LIN {X 0,Y 569.296,Z 343.315,A -85,B 0,C 180,E1 25931.653,E2 25931.653} C_VEL
LIN {X 0,Y 569.324,Z 343.315,A -85,B 0,C 180,E1 25928.382,E2 25928.382} C_VEL
LIN {X 0,Y 569.296,Z 343.305,A -85,B 0,C 180,E1 25925.543,E2 25925.543} C_VEL
LIN {X 0,Y 569.333,Z 343.299,A -85,B 0,C 180,E1 25922.315,E2 25922.315} C_VEL
LIN {X 0,Y 569.297,Z 343.304,A -85,B 0,C 180,E1 25919.396,E2 25919.396} C_VEL
LIN {X 0,Y 569.337,Z 343.298,A -85,B 0,C 180,E1 25916.173,E2 25916.173} C_VEL
LIN {X 0,Y 569.304,Z 343.315,A -85,B 0,C 180,E1 25913.141,E2 25913.141} C_VEL
LIN {X 0,Y 569.317,Z 343.31,A -85,B 0,C 180,E1 25909.782,E2 25909.782} C_VEL
LIN {X 0,Y 569.309,Z 343.253,A -85,B 0,C 180,E1 25906.802,E2 25906.802} C_VEL
LIN {X 0,Y 569.309,Z 343.313,A -85,B 0,C 180,E1 25903.47,E2 25903.47} C_VEL
LIN {X 0,Y 569.334,Z 343.255,A -85,B 0,C 180,E1 25900.4,E2 25900.4} C_VEL
LIN {X 0,Y 569.305,Z 343.303,A -85,B 0,C 180,E1 25897.226,E2 25897.226} C_VEL
LIN {X 0,Y 569.343,Z 343.264,A -85,B 0,C 180,E1 25894.18,E2 25894.18} C_VEL
LIN {X 0,Y 569.305,Z 343.306,A -85,B 0,C 180,E1 25891,E2 25891} C_VEL
LIN {X 0,Y 569.313,Z 343.38,A -85,B 0,C 180,E1 25890.889,E2 25890.889} C_VEL
LIN {X 0,Y 570.615,Z 346.769,A -85,B 0,C 180,E1 25890.271,E2 25890.271} C_VEL
LIN {X 0,Y 571.971,Z 348.701,A -85,B 0,C 180,E1 25889.828,E2 25889.828} C_VEL
LIN {X 0,Y 574.926,Z 352.956,A -85,B 0,C 180,E1 25889.248,E2 25889.248} C_VEL
LIN {X 0,Y 584.169,Z 364.72,A -85,B 0,C 180,E1 25887.634,E2 25887.634} C_VEL
LIN {X 0,Y 598.802,Z 384.338,A -85,B 0,C 180,E1 25885.262,E2 25885.262} C_VEL
LIN {X 0,Y 616.624,Z 409.316,A -85,B 0,C 180,E1 25882.622,E2 25882.622} C_VEL
LIN {X 0,Y 624.459,Z 421.118,A -85,B 0,C 180,E1 25881.519,E2 25881.519} C_VEL
LIN {X 0,Y 618.445,Z 624.42,A -85,B 0,C 180,E1 25878.613,E2 25878.613} C_VEL
LIN {X 0,Y 612.62,Z 826.414,A -85,B 0,C 180,E1 25875.768,E2 25875.768} C_VEL
LIN {X 0,Y 611.271,Z 850.143,A -85,B 0,C 180,E1 25875.338,E2 25875.338} C_VEL
LIN {X 0,Y 609.033,Z 878.867,A -85,B 0,C 180,E1 25874.632,E2 25874.632} C_VEL
LIN {X 0,Y 606.973,Z 900.534,A -85,B 0,C 180,E1 25873.955,E2 25873.955} C_VEL
LIN {X 0,Y 604.712,Z 921.393,A -85,B 0,C 180,E1 25873.181,E2 25873.181} C_VEL
LIN {X 0,Y 602.472,Z 940.413,A -85,B 0,C 180,E1 25872.36,E2 25872.36} C_VEL
LIN {X 0,Y 599.944,Z 959.81,A -85,B 0,C 180,E1 25871.41,E2 25871.41} C_VEL
LIN {X 0,Y 597.096,Z 980.312,A -85,B 0,C 180,E1 25870.268,E2 25870.268} C_VEL
LIN {X 0,Y 593.449,Z 1004.907,A -85,B 0,C 180,E1 25868.687,E2 25868.687} C_VEL
LIN {X 0,Y 590.181,Z 1025.558,A -85,B 0,C 180,E1 25867.154,E2 25867.154} C_VEL
LIN {X 0,Y 587.381,Z 1042.97,A -85,B 0,C 180,E1 25865.709,E2 25865.709} C_VEL
LIN {X 0,Y 584.6,Z 1060.165,A -85,B 0,C 180,E1 25864.124,E2 25864.124} C_VEL
LIN {X 0,Y 581.463,Z 1079.875,A -85,B 0,C 180,E1 25862.096,E2 25862.096} C_VEL
LIN {X 0,Y 578.616,Z 1097.987,A -85,B 0,C 180,E1 25859.96,E2 25859.96} C_VEL
LIN {X 0,Y 576.364,Z 1112.967,A -85,B 0,C 180,E1 25857.99,E2 25857.99} C_VEL
LIN {X 0,Y 574.256,Z 1127.882,A -85,B 0,C 180,E1 25855.803,E2 25855.803} C_VEL
LIN {X 0,Y 572.235,Z 1143.703,A -85,B 0,C 180,E1 25853.15,E2 25853.15} C_VEL
LIN {X 0,Y 570.92,Z 1155.266,A -85,B 0,C 180,E1 25850.932,E2 25850.932} C_VEL
LIN {X 0,Y 569.924,Z 1165.445,A -85,B 0,C 180,E1 25848.726,E2 25848.726} C_VEL
LIN {X 0,Y 569.029,Z 1176.304,A -85,B 0,C 180,E1 25846.015,E2 25846.015} C_VEL
LIN {X 0,Y 568.479,Z 1185.17,A -85,B 0,C 180,E1 25843.321,E2 25843.321} C_VEL
LIN {X 0,Y 568.159,Z 1191.597,A -85,B 0,C 180,E1 25840.956,E2 25840.956} C_VEL
LIN {X 0,Y 568.007,Z 1197.191,A -85,B 0,C 180,E1 25838.381,E2 25838.381} C_VEL
LIN {X 0,Y 567.933,Z 1201.538,A -85,B 0,C 180,E1 25835.557,E2 25835.557} C_VEL
LIN {X 0,Y 567.917,Z 1203.848,A -85,B 0,C 180,E1 25833.129,E2 25833.129} C_VEL
LIN {X 0,Y 567.906,Z 1204.804,A -85,B 0,C 180,E1 25830.908,E2 25830.908} C_VEL
LIN {X 0,Y 567.916,Z 1204.736,A -85,B 0,C 180,E1 25828.789,E2 25828.789} C_VEL
LIN {X 0,Y 567.912,Z 1203.507,A -85,B 0,C 180,E1 25826.366,E2 25826.366} C_VEL
LIN {X 0,Y 567.948,Z 1200.336,A -85,B 0,C 180,E1 25823.531,E2 25823.531} C_VEL
LIN {X 0,Y 568.029,Z 1196.126,A -85,B 0,C 180,E1 25821.089,E2 25821.089} C_VEL
LIN {X 0,Y 568.191,Z 1190.834,A -85,B 0,C 180,E1 25818.736,E2 25818.736} C_VEL
LIN {X 0,Y 568.577,Z 1183.471,A -85,B 0,C 180,E1 25816.106,E2 25816.106} C_VEL
LIN {X 0,Y 569.205,Z 1173.921,A -85,B 0,C 180,E1 25813.362,E2 25813.362} C_VEL
LIN {X 0,Y 570.006,Z 1164.53,A -85,B 0,C 180,E1 25811.064,E2 25811.064} C_VEL
LIN {X 0,Y 571.043,Z 1154.241,A -85,B 0,C 180,E1 25808.857,E2 25808.857} C_VEL
LIN {X 0,Y 572.616,Z 1140.8,A -85,B 0,C 180,E1 25806.321,E2 25806.321} C_VEL
LIN {X 0,Y 574.531,Z 1125.781,A -85,B 0,C 180,E1 25803.877,E2 25803.877} C_VEL
LIN {X 0,Y 576.537,Z 1111.839,A -85,B 0,C 180,E1 25801.854,E2 25801.854} C_VEL
LIN {X 0,Y 579.026,Z 1095.326,A -85,B 0,C 180,E1 25799.704,E2 25799.704} C_VEL
LIN {X 0,Y 582.167,Z 1075.37,A -85,B 0,C 180,E1 25797.428,E2 25797.428} C_VEL
LIN {X 0,Y 584.781,Z 1059.05,A -85,B 0,C 180,E1 25795.77,E2 25795.77} C_VEL
LIN {X 0,Y 587.479,Z 1042.377,A -85,B 0,C 180,E1 25794.24,E2 25794.24} C_VEL
LIN {X 0,Y 590.375,Z 1024.364,A -85,B 0,C 180,E1 25792.752,E2 25792.752} C_VEL
LIN {X 0,Y 594.048,Z 1001.028,A -85,B 0,C 180,E1 25791.044,E2 25791.044} C_VEL
LIN {X 0,Y 597.217,Z 979.404,A -85,B 0,C 180,E1 25789.679,E2 25789.679} C_VEL
LIN {X 0,Y 599.973,Z 959.579,A -85,B 0,C 180,E1 25788.578,E2 25788.578} C_VEL
LIN {X 0,Y 602.469,Z 940.393,A -85,B 0,C 180,E1 25787.639,E2 25787.639} C_VEL
LIN {X 0,Y 604.747,Z 921.017,A -85,B 0,C 180,E1 25786.805,E2 25786.805} C_VEL
LIN {X 0,Y 607.067,Z 899.553,A -85,B 0,C 180,E1 25786.013,E2 25786.013} C_VEL
LIN {X 0,Y 609.581,Z 872.863,A -85,B 0,C 180,E1 25785.2,E2 25785.2} C_VEL
LIN {X 0,Y 611.435,Z 847.126,A -85,B 0,C 180,E1 25784.602,E2 25784.602} C_VEL
LIN {X 0,Y 612.671,Z 825.024,A -85,B 0,C 180,E1 25784.212,E2 25784.212} C_VEL
LIN {X 0,Y 618.765,Z 612.923,A -85,B 0,C 180,E1 25781.224,E2 25781.224} C_VEL
LIN {X 0,Y 624.762,Z 420.905,A -85,B 0,C 180,E1 25778.456,E2 25778.456} C_VEL
LIN {X 0,Y 613.339,Z 403.227,A -85,B 0,C 180,E1 25776.668,E2 25776.668} C_VEL
LIN {X 0,Y 604.018,Z 389.622,A -85,B 0,C 180,E1 25775.088,E2 25775.088} C_VEL
LIN {X 0,Y 597.282,Z 380.633,A -85,B 0,C 180,E1 25773.881,E2 25773.881} C_VEL
LIN {X 0,Y 592.482,Z 374.303,A -85,B 0,C 180,E1 25772.974,E2 25772.974} C_VEL
LIN {X 0,Y 588.914,Z 369.679,A -85,B 0,C 180,E1 25772.274,E2 25772.274} C_VEL
LIN {X 0,Y 581.287,Z 359.993,A -85,B 0,C 180,E1 25770.694,E2 25770.694} C_VEL
LIN {X 0,Y 577.779,Z 355.627,A -85,B 0,C 180,E1 25769.923,E2 25769.923} C_VEL
LIN {X 0,Y 576.035,Z 353.726,A -85,B 0,C 180,E1 25769.536,E2 25769.536} C_VEL
LIN {X 0,Y 572.86,Z 349.891,A -85,B 0,C 180,E1 25768.799,E2 25768.799} C_VEL
LIN {X 0,Y 571.886,Z 348.208,A -85,B 0,C 180,E1 25768.51,E2 25768.51} C_VEL
LIN {X 0,Y 569.602,Z 344.596,A -85,B 0,C 180,E1 25767.495,E2 25767.495} C_VEL
LIN {X 0,Y 569.31,Z 343.269,A -85,B 0,C 180,E1 25767.171,E2 25767.171} C_VEL
LIN {X 0,Y 569.38,Z 343.289,A -85,B 0,C 180,E1 25764.043,E2 25764.043} C_VEL
LIN {X 0,Y 569.313,Z 343.291,A -85,B 0,C 180,E1 25760.881,E2 25760.881} C_VEL
LIN {X 0,Y 569.371,Z 343.26,A -85,B 0,C 180,E1 25757.687,E2 25757.687} C_VEL
LIN {X 0,Y 569.319,Z 343.314,A -85,B 0,C 180,E1 25754.546,E2 25754.546} C_VEL
LIN {X 0,Y 569.347,Z 343.269,A -85,B 0,C 180,E1 25751.241,E2 25751.241} C_VEL
LIN {X 0,Y 569.32,Z 343.289,A -85,B 0,C 180,E1 25748.28,E2 25748.28} C_VEL
LIN {X 0,Y 569.338,Z 343.294,A -85,B 0,C 180,E1 25744.937,E2 25744.937} C_VEL
LIN {X 0,Y 569.33,Z 343.268,A -85,B 0,C 180,E1 25741.912,E2 25741.912} C_VEL
LIN {X 0,Y 569.33,Z 343.315,A -85,B 0,C 180,E1 25738.591,E2 25738.591} C_VEL
LIN {X 0,Y 569.357,Z 343.259,A -85,B 0,C 180,E1 25735.467,E2 25735.467} C_VEL
LIN {X 0,Y 569.322,Z 343.3,A -85,B 0,C 180,E1 25732.228,E2 25732.228} C_VEL
LIN {X 0,Y 569.379,Z 343.279,A -85,B 0,C 180,E1 25729,E2 25729} C_VEL
LIN {X 0,Y 569.319,Z 343.267,A -85,B 0,C 180,E1 25725.799,E2 25725.799} C_VEL
LIN {X 0,Y 569.368,Z 343.301,A -85,B 0,C 180,E1 25722.524,E2 25722.524} C_VEL
LIN {X 0,Y 569.329,Z 343.284,A -85,B 0,C 180,E1 25719.399,E2 25719.399} C_VEL
LIN {X 0,Y 569.392,Z 343.421,A -85,B 0,C 180,E1 25718.9,E2 25718.9} C_VEL
LIN {X 0,Y 570.358,Z 346.246,A -85,B 0,C 180,E1 25718.614,E2 25718.614} C_VEL
LIN {X 0,Y 572.684,Z 348.869,A -85,B 0,C 180,E1 25718.06,E2 25718.06} C_VEL
LIN {X 0,Y 574.711,Z 350.146,A -85,B 0,C 180,E1 25717.617,E2 25717.617} C_VEL
LIN {X 0,Y 576.858,Z 353.718,A -85,B 0,C 180,E1 25717.099,E2 25717.099} C_VEL
LIN {X 0,Y 580.018,Z 356.535,A -85,B 0,C 180,E1 25716.425,E2 25716.425} C_VEL
LIN {X 0,Y 582.778,Z 360.473,A -85,B 0,C 180,E1 25715.818,E2 25715.818} C_VEL
LIN {X 0,Y 585.289,Z 362.868,A -85,B 0,C 180,E1 25715.311,E2 25715.311} C_VEL
LIN {X 0,Y 588.636,Z 367.172,A -85,B 0,C 180,E1 25714.628,E2 25714.628} C_VEL
LIN {X 0,Y 597.326,Z 377.95,A -85,B 0,C 180,E1 25712.969,E2 25712.969} C_VEL
LIN {X 0,Y 608.831,Z 393.554,A -85,B 0,C 180,E1 25710.941,E2 25710.941} C_VEL
LIN {X 0,Y 620.103,Z 410.5,A -85,B 0,C 180,E1 25709.111,E2 25709.111} C_VEL
LIN {X 0,Y 624.682,Z 417.785,A -85,B 0,C 180,E1 25708.41,E2 25708.41} C_VEL
LIN {X 0,Y 618.203,Z 625.916,A -85,B 0,C 180,E1 25705.412,E2 25705.412} C_VEL
LIN {X 0,Y 614.777,Z 746.22,A -85,B 0,C 180,E1 25703.721,E2 25703.721} C_VEL
LIN {X 0,Y 613.881,Z 753.921,A -85,B 0,C 180,E1 25703.681,E2 25703.681} C_VEL
LIN {X 0,Y 608.994,Z 774.548,A -85,B 0,C 180,E1 25703.822,E2 25703.822} C_VEL
LIN {X 0,Y 608.288,Z 781.156,A -85,B 0,C 180,E1 25703.781,E2 25703.781} C_VEL
LIN {X 0,Y 606.727,Z 825.165,A -85,B 0,C 180,E1 25703.134,E2 25703.134} C_VEL
LIN {X 0,Y 604.843,Z 852.015,A -85,B 0,C 180,E1 25702.575,E2 25702.575} C_VEL
LIN {X 0,Y 602.85,Z 874.745,A -85,B 0,C 180,E1 25701.965,E2 25701.965} C_VEL
LIN {X 0,Y 600.188,Z 900.951,A -85,B 0,C 180,E1 25701.092,E2 25701.092} C_VEL
LIN {X 0,Y 597.063,Z 926.428,A -85,B 0,C 180,E1 25700.042,E2 25700.042} C_VEL
LIN {X 0,Y 593.864,Z 950.106,A -85,B 0,C 180,E1 25698.888,E2 25698.888} C_VEL
LIN {X 0,Y 590.327,Z 973.89,A -85,B 0,C 180,E1 25697.529,E2 25697.529} C_VEL
LIN {X 0,Y 587.148,Z 993.791,A -85,B 0,C 180,E1 25696.222,E2 25696.222} C_VEL
LIN {X 0,Y 583.963,Z 1013.149,A -85,B 0,C 180,E1 25694.794,E2 25694.794} C_VEL
LIN {X 0,Y 580.163,Z 1035.792,A -85,B 0,C 180,E1 25692.902,E2 25692.902} C_VEL
LIN {X 0,Y 576.836,Z 1055.052,A -85,B 0,C 180,E1 25691.059,E2 25691.059} C_VEL
LIN {X 0,Y 573.849,Z 1072.78,A -85,B 0,C 180,E1 25689.16,E2 25689.16} C_VEL
LIN {X 0,Y 570.546,Z 1092.991,A -85,B 0,C 180,E1 25686.697,E2 25686.697} C_VEL
LIN {X 0,Y 568.077,Z 1108.692,A -85,B 0,C 180,E1 25684.523,E2 25684.523} C_VEL
LIN {X 0,Y 565.787,Z 1124.739,A -85,B 0,C 180,E1 25682.016,E2 25682.016} C_VEL
LIN {X 0,Y 563.914,Z 1138.861,A -85,B 0,C 180,E1 25679.47,E2 25679.47} C_VEL
LIN {X 0,Y 562.473,Z 1151.648,A -85,B 0,C 180,E1 25676.841,E2 25676.841} C_VEL
LIN {X 0,Y 561.38,Z 1163.044,A -85,B 0,C 180,E1 25674.071,E2 25674.071} C_VEL
LIN {X 0,Y 560.732,Z 1171.84,A -85,B 0,C 180,E1 25671.551,E2 25671.551} C_VEL
LIN {X 0,Y 560.291,Z 1179.722,A -85,B 0,C 180,E1 25668.844,E2 25668.844} C_VEL
LIN {X 0,Y 560.05,Z 1185.816,A -85,B 0,C 180,E1 25666.152,E2 25666.152} C_VEL
LIN {X 0,Y 559.953,Z 1189.82,A -85,B 0,C 180,E1 25663.844,E2 25663.844} C_VEL
LIN {X 0,Y 559.917,Z 1192.912,A -85,B 0,C 180,E1 25661.328,E2 25661.328} C_VEL
LIN {X 0,Y 559.909,Z 1194.644,A -85,B 0,C 180,E1 25658.627,E2 25658.627} C_VEL
LIN {X 0,Y 559.913,Z 1194.855,A -85,B 0,C 180,E1 25656.254,E2 25656.254} C_VEL
LIN {X 0,Y 559.91,Z 1193.988,A -85,B 0,C 180,E1 25653.994,E2 25653.994} C_VEL
LIN {X 0,Y 559.923,Z 1191.789,A -85,B 0,C 180,E1 25651.535,E2 25651.535} C_VEL
LIN {X 0,Y 560.002,Z 1187.772,A -85,B 0,C 180,E1 25648.772,E2 25648.772} C_VEL
LIN {X 0,Y 560.145,Z 1182.479,A -85,B 0,C 180,E1 25646.213,E2 25646.213} C_VEL
LIN {X 0,Y 560.447,Z 1176.363,A -85,B 0,C 180,E1 25643.855,E2 25643.855} C_VEL
LIN {X 0,Y 560.961,Z 1168.311,A -85,B 0,C 180,E1 25641.286,E2 25641.286} C_VEL
LIN {X 0,Y 561.873,Z 1157.755,A -85,B 0,C 180,E1 25638.504,E2 25638.504} C_VEL
LIN {X 0,Y 562.987,Z 1146.754,A -85,B 0,C 180,E1 25636.023,E2 25636.023} C_VEL
LIN {X 0,Y 564.674,Z 1132.973,A -85,B 0,C 180,E1 25633.331,E2 25633.331} C_VEL
LIN {X 0,Y 566.562,Z 1118.874,A -85,B 0,C 180,E1 25630.945,E2 25630.945} C_VEL
LIN {X 0,Y 568.991,Z 1103.007,A -85,B 0,C 180,E1 25628.561,E2 25628.561} C_VEL
LIN {X 0,Y 571.836,Z 1084.833,A -85,B 0,C 180,E1 25626.178,E2 25626.178} C_VEL
LIN {X 0,Y 574.666,Z 1067.976,A -85,B 0,C 180,E1 25624.217,E2 25624.217} C_VEL
LIN {X 0,Y 578.197,Z 1047.445,A -85,B 0,C 180,E1 25622.091,E2 25622.091} C_VEL
LIN {X 0,Y 581.602,Z 1027.065,A -85,B 0,C 180,E1 25620.25,E2 25620.25} C_VEL
LIN {X 0,Y 584.696,Z 1008.633,A -85,B 0,C 180,E1 25618.766,E2 25618.766} C_VEL
LIN {X 0,Y 588.482,Z 985.63,A -85,B 0,C 180,E1 25617.123,E2 25617.123} C_VEL
LIN {X 0,Y 591.988,Z 962.709,A -85,B 0,C 180,E1 25615.718,E2 25615.718} C_VEL
LIN {X 0,Y 595.353,Z 939.327,A -85,B 0,C 180,E1 25614.473,E2 25614.473} C_VEL
LIN {X 0,Y 598.747,Z 912.783,A -85,B 0,C 180,E1 25613.282,E2 25613.282} C_VEL
LIN {X 0,Y 601.432,Z 889.096,A -85,B 0,C 180,E1 25612.402,E2 25612.402} C_VEL
LIN {X 0,Y 604.11,Z 861.148,A -85,B 0,C 180,E1 25611.56,E2 25611.56} C_VEL
LIN {X 0,Y 605.996,Z 835.793,A -85,B 0,C 180,E1 25610.979,E2 25610.979} C_VEL
LIN {X 0,Y 607.3,Z 812.342,A -85,B 0,C 180,E1 25610.575,E2 25610.575} C_VEL
LIN {X 0,Y 613.778,Z 596.837,A -85,B 0,C 180,E1 25607.52,E2 25607.52} C_VEL
LIN {X 0,Y 619.14,Z 421.569,A -85,B 0,C 180,E1 25604.997,E2 25604.997} C_VEL
LIN {X 0,Y 605.811,Z 402.395,A -85,B 0,C 180,E1 25603.07,E2 25603.07} C_VEL
LIN {X 0,Y 589.286,Z 379.992,A -85,B 0,C 180,E1 25600.5,E2 25600.5} C_VEL
LIN {X 0,Y 583.743,Z 372.893,A -85,B 0,C 180,E1 25599.583,E2 25599.583} C_VEL
LIN {X 0,Y 579.056,Z 367.062,A -85,B 0,C 180,E1 25598.784,E2 25598.784} C_VEL
LIN {X 0,Y 575.08,Z 362.1,A -85,B 0,C 180,E1 25598.083,E2 25598.083} C_VEL
LIN {X 0,Y 571.76,Z 358.178,A -85,B 0,C 180,E1 25597.487,E2 25597.487} C_VEL
LIN {X 0,Y 570.576,Z 356.419,A -85,B 0,C 180,E1 25597.262,E2 25597.262} C_VEL
LIN {X 0,Y 567.534,Z 353.373,A -85,B 0,C 180,E1 25596.709,E2 25596.709} C_VEL
LIN {X 0,Y 565.807,Z 350.517,A -85,B 0,C 180,E1 25596.363,E2 25596.363} C_VEL
LIN {X 0,Y 563.016,Z 348.232,A -85,B 0,C 180,E1 25595.847,E2 25595.847} C_VEL
LIN {X 0,Y 561.6,Z 345.253,A -85,B 0,C 180,E1 25595.537,E2 25595.537} C_VEL
LIN {X 0,Y 561.418,Z 344.297,A -85,B 0,C 180,E1 25595.455,E2 25595.455} C_VEL
LIN {X 0,Y 561.348,Z 344.296,A -85,B 0,C 180,E1 25592.301,E2 25592.301} C_VEL
LIN {X 0,Y 561.394,Z 344.257,A -85,B 0,C 180,E1 25589.094,E2 25589.094} C_VEL
LIN {X 0,Y 561.35,Z 344.276,A -85,B 0,C 180,E1 25586.102,E2 25586.102} C_VEL
LIN {X 0,Y 561.384,Z 344.252,A -85,B 0,C 180,E1 25582.848,E2 25582.848} C_VEL
LIN {X 0,Y 561.354,Z 344.274,A -85,B 0,C 180,E1 25579.873,E2 25579.873} C_VEL
LIN {X 0,Y 561.376,Z 344.289,A -85,B 0,C 180,E1 25576.558,E2 25576.558} C_VEL
LIN {X 0,Y 561.357,Z 344.293,A -85,B 0,C 180,E1 25573.704,E2 25573.704} C_VEL
LIN {X 0,Y 561.375,Z 344.29,A -85,B 0,C 180,E1 25570.364,E2 25570.364} C_VEL
LIN {X 0,Y 561.37,Z 344.302,A -85,B 0,C 180,E1 25567.368,E2 25567.368} C_VEL
LIN {X 0,Y 561.364,Z 344.302,A -85,B 0,C 180,E1 25563.983,E2 25563.983} C_VEL
LIN {X 0,Y 561.411,Z 344.302,A -85,B 0,C 180,E1 25560.816,E2 25560.816} C_VEL
LIN {X 0,Y 561.359,Z 344.304,A -85,B 0,C 180,E1 25557.652,E2 25557.652} C_VEL
LIN {X 0,Y 561.43,Z 344.289,A -85,B 0,C 180,E1 25554.481,E2 25554.481} C_VEL
LIN {X 0,Y 561.357,Z 344.296,A -85,B 0,C 180,E1 25551.395,E2 25551.395} C_VEL
LIN {X 0,Y 561.424,Z 344.248,A -85,B 0,C 180,E1 25548.286,E2 25548.286} C_VEL
LIN {X 0,Y 561.358,Z 344.279,A -85,B 0,C 180,E1 25545.138,E2 25545.138} C_VEL
LIN {X 0,Y 561.422,Z 344.25,A -85,B 0,C 180,E1 25541.993,E2 25541.993} C_VEL
LIN {X 0,Y 561.362,Z 344.283,A -85,B 0,C 180,E1 25538.912,E2 25538.912} C_VEL
LIN {X 0,Y 561.415,Z 344.242,A -85,B 0,C 180,E1 25535.762,E2 25535.762} C_VEL
LIN {X 0,Y 561.371,Z 344.306,A -85,B 0,C 180,E1 25532.643,E2 25532.643} C_VEL
LIN {X 0,Y 561.43,Z 344.387,A -85,B 0,C 180,E1 25532.07,E2 25532.07} C_VEL
LIN {X 0,Y 562.942,Z 348.123,A -85,B 0,C 180,E1 25531.342,E2 25531.342} C_VEL
LIN {X 0,Y 564.329,Z 349.877,A -85,B 0,C 180,E1 25531,E2 25531} C_VEL
LIN {X 0,Y 567.386,Z 353.997,A -85,B 0,C 180,E1 25530.404,E2 25530.404} C_VEL
LIN {X 0,Y 569.176,Z 356.02,A -85,B 0,C 180,E1 25530.072,E2 25530.072} C_VEL
LIN {X 0,Y 572.752,Z 360.564,A -85,B 0,C 180,E1 25529.41,E2 25529.41} C_VEL
LIN {X 0,Y 585.685,Z 377.689,A -85,B 0,C 180,E1 25527.148,E2 25527.148} C_VEL
LIN {X 0,Y 599.12,Z 396.051,A -85,B 0,C 180,E1 25524.992,E2 25524.992} C_VEL
LIN {X 0,Y 615.081,Z 418.695,A -85,B 0,C 180,E1 25522.629,E2 25522.629} C_VEL
LIN {X 0,Y 619.245,Z 425.185,A -85,B 0,C 180,E1 25522.033,E2 25522.033} C_VEL
LIN {X 0,Y 612.96,Z 630.441,A -85,B 0,C 180,E1 25519.089,E2 25519.089} C_VEL
LIN {X 0,Y 607.03,Z 826.34,A -85,B 0,C 180,E1 25516.31,E2 25516.31} C_VEL
LIN {X 0,Y 605.619,Z 850.131,A -85,B 0,C 180,E1 25515.878,E2 25515.878} C_VEL
LIN {X 0,Y 603.276,Z 878.948,A -85,B 0,C 180,E1 25515.166,E2 25515.166} C_VEL
LIN {X 0,Y 601.061,Z 901.163,A -85,B 0,C 180,E1 25514.466,E2 25514.466} C_VEL
LIN {X 0,Y 598.683,Z 922.092,A -85,B 0,C 180,E1 25513.682,E2 25513.682} C_VEL
LIN {X 0,Y 596.29,Z 941.427,A -85,B 0,C 180,E1 25512.839,E2 25512.839} C_VEL
LIN {X 0,Y 593.544,Z 961.487,A -85,B 0,C 180,E1 25511.842,E2 25511.842} C_VEL
LIN {X 0,Y 589.929,Z 986.315,A -85,B 0,C 180,E1 25510.419,E2 25510.419} C_VEL
LIN {X 0,Y 586.377,Z 1008.494,A -85,B 0,C 180,E1 25508.934,E2 25508.934} C_VEL
LIN {X 0,Y 583.451,Z 1026.223,A -85,B 0,C 180,E1 25507.595,E2 25507.595} C_VEL
LIN {X 0,Y 580.646,Z 1042.828,A -85,B 0,C 180,E1 25506.202,E2 25506.202} C_VEL
LIN {X 0,Y 577.785,Z 1059.605,A -85,B 0,C 180,E1 25504.643,E2 25504.643} C_VEL
LIN {X 0,Y 574.6,Z 1078.508,A -85,B 0,C 180,E1 25502.687,E2 25502.687} C_VEL
LIN {X 0,Y 571.336,Z 1097.985,A -85,B 0,C 180,E1 25500.382,E2 25500.382} C_VEL
LIN {X 0,Y 569.021,Z 1112.608,A -85,B 0,C 180,E1 25498.437,E2 25498.437} C_VEL
LIN {X 0,Y 566.887,Z 1126.667,A -85,B 0,C 180,E1 25496.359,E2 25496.359} C_VEL
LIN {X 0,Y 564.719,Z 1142.547,A -85,B 0,C 180,E1 25493.698,E2 25493.698} C_VEL
LIN {X 0,Y 563.223,Z 1154.749,A -85,B 0,C 180,E1 25491.341,E2 25491.341} C_VEL
LIN {X 0,Y 562.124,Z 1164.984,A -85,B 0,C 180,E1 25489.104,E2 25489.104} C_VEL
LIN {X 0,Y 561.248,Z 1174.731,A -85,B 0,C 180,E1 25486.668,E2 25486.668} C_VEL
LIN {X 0,Y 560.562,Z 1184.561,A -85,B 0,C 180,E1 25483.723,E2 25483.723} C_VEL
LIN {X 0,Y 560.206,Z 1191.085,A -85,B 0,C 180,E1 25481.322,E2 25481.322} C_VEL
LIN {X 0,Y 560.034,Z 1196.331,A -85,B 0,C 180,E1 25478.936,E2 25478.936} C_VEL
LIN {X 0,Y 559.945,Z 1200.782,A -85,B 0,C 180,E1 25476.253,E2 25476.253} C_VEL
LIN {X 0,Y 559.914,Z 1203.641,A -85,B 0,C 180,E1 25473.481,E2 25473.481} C_VEL
LIN {X 0,Y 559.916,Z 1204.736,A -85,B 0,C 180,E1 25471.228,E2 25471.228} C_VEL
LIN {X 0,Y 559.906,Z 1204.804,A -85,B 0,C 180,E1 25469.079,E2 25469.079} C_VEL
LIN {X 0,Y 559.917,Z 1203.845,A -85,B 0,C 180,E1 25466.827,E2 25466.827} C_VEL
LIN {X 0,Y 559.933,Z 1201.534,A -85,B 0,C 180,E1 25464.364,E2 25464.364} C_VEL
LIN {X 0,Y 560.018,Z 1197.151,A -85,B 0,C 180,E1 25461.478,E2 25461.478} C_VEL
LIN {X 0,Y 560.181,Z 1191.594,A -85,B 0,C 180,E1 25458.886,E2 25458.886} C_VEL
LIN {X 0,Y 560.532,Z 1185.077,A -85,B 0,C 180,E1 25456.456,E2 25456.456} C_VEL
LIN {X 0,Y 561.163,Z 1175.941,A -85,B 0,C 180,E1 25453.649,E2 25453.649} C_VEL
LIN {X 0,Y 562.082,Z 1165.446,A -85,B 0,C 180,E1 25451.002,E2 25451.002} C_VEL
LIN {X 0,Y 563.161,Z 1155.269,A -85,B 0,C 180,E1 25448.765,E2 25448.765} C_VEL
LIN {X 0,Y 564.639,Z 1143.132,A -85,B 0,C 180,E1 25446.409,E2 25446.409} C_VEL
LIN {X 0,Y 566.813,Z 1127.181,A -85,B 0,C 180,E1 25443.72,E2 25443.72} C_VEL
LIN {X 0,Y 569.021,Z 1112.608,A -85,B 0,C 180,E1 25441.563,E2 25441.563} C_VEL
LIN {X 0,Y 571.336,Z 1097.984,A -85,B 0,C 180,E1 25439.618,E2 25439.618} C_VEL
LIN {X 0,Y 574.6,Z 1078.508,A -85,B 0,C 180,E1 25437.313,E2 25437.313} C_VEL
LIN {X 0,Y 577.784,Z 1059.604,A -85,B 0,C 180,E1 25435.356,E2 25435.356} C_VEL
LIN {X 0,Y 580.645,Z 1042.823,A -85,B 0,C 180,E1 25433.798,E2 25433.798} C_VEL
LIN {X 0,Y 583.449,Z 1026.214,A -85,B 0,C 180,E1 25432.405,E2 25432.405} C_VEL
LIN {X 0,Y 586.487,Z 1007.817,A -85,B 0,C 180,E1 25431.018,E2 25431.018} C_VEL
LIN {X 0,Y 590.301,Z 983.795,A -85,B 0,C 180,E1 25429.427,E2 25429.427} C_VEL
LIN {X 0,Y 593.652,Z 960.624,A -85,B 0,C 180,E1 25428.113,E2 25428.113} C_VEL
LIN {X 0,Y 596.285,Z 941.391,A -85,B 0,C 180,E1 25427.161,E2 25427.161} C_VEL
LIN {X 0,Y 598.672,Z 922.084,A -85,B 0,C 180,E1 25426.319,E2 25426.319} C_VEL
LIN {X 0,Y 601.049,Z 901.154,A -85,B 0,C 180,E1 25425.535,E2 25425.535} C_VEL
LIN {X 0,Y 603.272,Z 878.878,A -85,B 0,C 180,E1 25424.834,E2 25424.834} C_VEL
LIN {X 0,Y 605.602,Z 850.195,A -85,B 0,C 180,E1 25424.125,E2 25424.125} C_VEL
LIN {X 0,Y 607.019,Z 826.32,A -85,B 0,C 180,E1 25423.691,E2 25423.691} C_VEL
LIN {X 0,Y 613.57,Z 611.894,A -85,B 0,C 180,E1 25420.642,E2 25420.642} C_VEL
LIN {X 0,Y 619.771,Z 424.932,A -85,B 0,C 180,E1 25417.921,E2 25417.921} C_VEL
LIN {X 0,Y 609.225,Z 408.462,A -85,B 0,C 180,E1 25416.218,E2 25416.218} C_VEL
LIN {X 0,Y 600.547,Z 395.741,A -85,B 0,C 180,E1 25414.71,E2 25414.71} C_VEL
LIN {X 0,Y 593.903,Z 386.796,A -85,B 0,C 180,E1 25413.491,E2 25413.491} C_VEL
LIN {X 0,Y 586.761,Z 377.199,A -85,B 0,C 180,E1 25412.09,E2 25412.09} C_VEL
LIN {X 0,Y 578.347,Z 366.644,A -85,B 0,C 180,E1 25410.32,E2 25410.32} C_VEL
LIN {X 0,Y 574.092,Z 361.286,A -85,B 0,C 180,E1 25409.36,E2 25409.36} C_VEL
LIN {X 0,Y 570.538,Z 357.103,A -85,B 0,C 180,E1 25408.527,E2 25408.527} C_VEL
LIN {X 0,Y 569.215,Z 355.274,A -85,B 0,C 180,E1 25408.199,E2 25408.199} C_VEL
LIN {X 0,Y 565.611,Z 351.285,A -85,B 0,C 180,E1 25407.306,E2 25407.306} C_VEL
LIN {X 0,Y 564.351,Z 349.548,A -85,B 0,C 180,E1 25406.973,E2 25406.973} C_VEL
LIN {X 0,Y 562.536,Z 347.462,A -85,B 0,C 180,E1 25406.383,E2 25406.383} C_VEL
LIN {X 0,Y 561.397,Z 344.277,A -85,B 0,C 180,E1 25405.532,E2 25405.532} C_VEL
LIN {X 0,Y 561.387,Z 344.253,A -85,B 0,C 180,E1 25402.516,E2 25402.516} C_VEL
LIN {X 0,Y 561.382,Z 344.284,A -85,B 0,C 180,E1 25399.131,E2 25399.131} C_VEL
LIN {X 0,Y 561.435,Z 344.27,A -85,B 0,C 180,E1 25395.912,E2 25395.912} C_VEL
LIN {X 0,Y 561.373,Z 344.255,A -85,B 0,C 180,E1 25392.76,E2 25392.76} C_VEL
LIN {X 0,Y 561.443,Z 344.297,A -85,B 0,C 180,E1 25389.534,E2 25389.534} C_VEL
LIN {X 0,Y 561.374,Z 344.252,A -85,B 0,C 180,E1 25386.34,E2 25386.34} C_VEL
LIN {X 0,Y 561.417,Z 344.283,A -85,B 0,C 180,E1 25383.063,E2 25383.063} C_VEL
LIN {X 0,Y 561.385,Z 344.266,A -85,B 0,C 180,E1 25380,E2 25380} C_VEL
LIN {X 0,Y 561.392,Z 344.256,A -85,B 0,C 180,E1 25376.63,E2 25376.63} C_VEL
LIN {X 0,Y 561.419,Z 344.296,A -85,B 0,C 180,E1 25373.455,E2 25373.455} C_VEL
LIN {X 0,Y 561.379,Z 344.253,A -85,B 0,C 180,E1 25370.155,E2 25370.155} C_VEL
LIN {X 0,Y 561.444,Z 344.271,A -85,B 0,C 180,E1 25366.928,E2 25366.928} C_VEL
LIN {X 0,Y 561.384,Z 344.28,A -85,B 0,C 180,E1 25363.737,E2 25363.737} C_VEL
LIN {X 0,Y 561.466,Z 344.455,A -85,B 0,C 180,E1 25360.642,E2 25360.642} C_VEL
LIN {X 0,Y 562.483,Z 347.372,A -85,B 0,C 180,E1 25360.314,E2 25360.314} C_VEL
LIN {X 0,Y 564.85,Z 349.912,A -85,B 0,C 180,E1 25359.699,E2 25359.699} C_VEL
LIN {X 0,Y 566.956,Z 351.173,A -85,B 0,C 180,E1 25359.197,E2 25359.197} C_VEL
LIN {X 0,Y 569.05,Z 354.816,A -85,B 0,C 180,E1 25358.644,E2 25358.644} C_VEL
LIN {X 0,Y 572.443,Z 357.771,A -85,B 0,C 180,E1 25357.861,E2 25357.861} C_VEL
LIN {X 0,Y 575.162,Z 361.595,A -85,B 0,C 180,E1 25357.217,E2 25357.217} C_VEL
LIN {X 0,Y 577.659,Z 363.959,A -85,B 0,C 180,E1 25356.675,E2 25356.675} C_VEL
LIN {X 0,Y 580.948,Z 368.225,A -85,B 0,C 180,E1 25355.953,E2 25355.953} C_VEL
LIN {X 0,Y 582.884,Z 370.237,A -85,B 0,C 180,E1 25355.553,E2 25355.553} C_VEL
LIN {X 0,Y 586.663,Z 374.812,A -85,B 0,C 180,E1 25354.78,E2 25354.78} C_VEL
LIN {X 0,Y 595.487,Z 386.286,A -85,B 0,C 180,E1 25353.067,E2 25353.067} C_VEL
LIN {X 0,Y 603.082,Z 396.644,A -85,B 0,C 180,E1 25351.694,E2 25351.694} C_VEL
LIN {X 0,Y 611.202,Z 408.426,A -85,B 0,C 180,E1 25350.312,E2 25350.312} C_VEL
LIN {X 0,Y 619.71,Z 421.852,A -85,B 0,C 180,E1 25348.943,E2 25348.943} C_VEL
LIN {X 0,Y 612.74,Z 632.307,A -85,B 0,C 180,E1 25345.887,E2 25345.887} C_VEL
LIN {X 0,Y 608.288,Z 781.156,A -85,B 0,C 180,E1 25343.781,E2 25343.781} C_VEL
LIN {X 0,Y 607.385,Z 788.857,A -85,B 0,C 180,E1 25343.742,E2 25343.742} C_VEL
LIN {X 0,Y 602.412,Z 809.467,A -85,B 0,C 180,E1 25343.883,E2 25343.883} C_VEL
LIN {X 0,Y 601.606,Z 816.058,A -85,B 0,C 180,E1 25343.829,E2 25343.829} C_VEL
LIN {X 0,Y 600.236,Z 838.718,A -85,B 0,C 180,E1 25343.423,E2 25343.423} C_VEL
LIN {X 0,Y 598.055,Z 865.986,A -85,B 0,C 180,E1 25342.771,E2 25342.771} C_VEL
LIN {X 0,Y 595.472,Z 890.985,A -85,B 0,C 180,E1 25341.991,E2 25341.991} C_VEL
LIN {X 0,Y 592.786,Z 913.646,A -85,B 0,C 180,E1 25341.136,E2 25341.136} C_VEL
LIN {X 0,Y 589.41,Z 939.136,A -85,B 0,C 180,E1 25339.988,E2 25339.988} C_VEL
LIN {X 0,Y 585.631,Z 964.205,A -85,B 0,C 180,E1 25338.642,E2 25338.642} C_VEL
LIN {X 0,Y 581.602,Z 988.997,A -85,B 0,C 180,E1 25337.084,E2 25337.084} C_VEL
LIN {X 0,Y 577.792,Z 1010.962,A -85,B 0,C 180,E1 25335.476,E2 25335.476} C_VEL
LIN {X 0,Y 574.072,Z 1032.233,A -85,B 0,C 180,E1 25333.711,E2 25333.711} C_VEL
LIN {X 0,Y 570.256,Z 1053.246,A -85,B 0,C 180,E1 25331.715,E2 25331.715} C_VEL
LIN {X 0,Y 567.142,Z 1070.621,A -85,B 0,C 180,E1 25329.854,E2 25329.854} C_VEL
LIN {X 0,Y 563.886,Z 1089.493,A -85,B 0,C 180,E1 25327.587,E2 25327.587} C_VEL
LIN {X 0,Y 561.039,Z 1106.318,A -85,B 0,C 180,E1 25325.269,E2 25325.269} C_VEL
LIN {X 0,Y 558.801,Z 1120.525,A -85,B 0,C 180,E1 25323.075,E2 25323.075} C_VEL
LIN {X 0,Y 556.666,Z 1135.627,A -85,B 0,C 180,E1 25320.432,E2 25320.432} C_VEL
LIN {X 0,Y 555.077,Z 1147.987,A -85,B 0,C 180,E1 25317.926,E2 25317.926} C_VEL
LIN {X 0,Y 553.834,Z 1159.653,A -85,B 0,C 180,E1 25315.218,E2 25315.218} C_VEL
LIN {X 0,Y 552.949,Z 1169.704,A -85,B 0,C 180,E1 25312.429,E2 25312.429} C_VEL
LIN {X 0,Y 552.454,Z 1177.038,A -85,B 0,C 180,E1 25310.002,E2 25310.002} C_VEL
LIN {X 0,Y 552.145,Z 1183.32,A -85,B 0,C 180,E1 25307.494,E2 25307.494} C_VEL
LIN {X 0,Y 551.986,Z 1188.869,A -85,B 0,C 180,E1 25304.583,E2 25304.583} C_VEL
LIN {X 0,Y 551.928,Z 1192.128,A -85,B 0,C 180,E1 25302.131,E2 25302.131} C_VEL
LIN {X 0,Y 551.912,Z 1194.151,A -85,B 0,C 180,E1 25299.7,E2 25299.7} C_VEL
LIN {X 0,Y 551.912,Z 1194.987,A -85,B 0,C 180,E1 25296.867,E2 25296.867} C_VEL
LIN {X 0,Y 551.911,Z 1194.116,A -85,B 0,C 180,E1 25294.156,E2 25294.156} C_VEL
LIN {X 0,Y 551.924,Z 1192.113,A -85,B 0,C 180,E1 25291.765,E2 25291.765} C_VEL
LIN {X 0,Y 551.985,Z 1188.636,A -85,B 0,C 180,E1 25289.17,E2 25289.17} C_VEL
LIN {X 0,Y 552.144,Z 1183.203,A -85,B 0,C 180,E1 25286.366,E2 25286.366} C_VEL
LIN {X 0,Y 552.457,Z 1176.936,A -85,B 0,C 180,E1 25283.87,E2 25283.87} C_VEL
LIN {X 0,Y 552.964,Z 1169.346,A -85,B 0,C 180,E1 25281.369,E2 25281.369} C_VEL
LIN {X 0,Y 553.942,Z 1158.618,A -85,B 0,C 180,E1 25278.442,E2 25278.442} C_VEL
LIN {X 0,Y 555.102,Z 1147.72,A -85,B 0,C 180,E1 25275.927,E2 25275.927} C_VEL
LIN {X 0,Y 556.785,Z 1134.687,A -85,B 0,C 180,E1 25273.302,E2 25273.302} C_VEL
LIN {X 0,Y 558.838,Z 1120.181,A -85,B 0,C 180,E1 25270.779,E2 25270.779} C_VEL
LIN {X 0,Y 561.24,Z 1105.154,A -85,B 0,C 180,E1 25268.47,E2 25268.47} C_VEL
LIN {X 0,Y 564.346,Z 1086.545,A -85,B 0,C 180,E1 25265.953,E2 25265.953} C_VEL
LIN {X 0,Y 567.285,Z 1069.842,A -85,B 0,C 180,E1 25263.968,E2 25263.968} C_VEL
LIN {X 0,Y 570.445,Z 1052.278,A -85,B 0,C 180,E1 25262.096,E2 25262.096} C_VEL
LIN {X 0,Y 574.488,Z 1029.652,A -85,B 0,C 180,E1 25259.975,E2 25259.975} C_VEL
LIN {X 0,Y 577.904,Z 1010.317,A -85,B 0,C 180,E1 25258.383,E2 25258.383} C_VEL
LIN {X 0,Y 581.783,Z 987.961,A -85,B 0,C 180,E1 25256.754,E2 25256.754} C_VEL
LIN {X 0,Y 585.706,Z 963.663,A -85,B 0,C 180,E1 25255.238,E2 25255.238} C_VEL
LIN {X 0,Y 589.514,Z 938.398,A -85,B 0,C 180,E1 25253.887,E2 25253.887} C_VEL
LIN {X 0,Y 592.877,Z 912.822,A -85,B 0,C 180,E1 25252.74,E2 25252.74} C_VEL
LIN {X 0,Y 595.61,Z 889.798,A -85,B 0,C 180,E1 25251.878,E2 25251.878} C_VEL
LIN {X 0,Y 598.41,Z 861.898,A -85,B 0,C 180,E1 25251.03,E2 25251.03} C_VEL
LIN {X 0,Y 600.372,Z 836.638,A -85,B 0,C 180,E1 25250.444,E2 25250.444} C_VEL
LIN {X 0,Y 601.704,Z 814.012,A -85,B 0,C 180,E1 25250.048,E2 25250.048} C_VEL
LIN {X 0,Y 608.226,Z 606.452,A -85,B 0,C 180,E1 25247.088,E2 25247.088} C_VEL
LIN {X 0,Y 613.982,Z 425.694,A -85,B 0,C 180,E1 25244.478,E2 25244.478} C_VEL
LIN {X 0,Y 601.772,Z 408.117,A -85,B 0,C 180,E1 25242.682,E2 25242.682} C_VEL
LIN {X 0,Y 584.512,Z 384.458,A -85,B 0,C 180,E1 25239.935,E2 25239.935} C_VEL
LIN {X 0,Y 575.771,Z 373.571,A -85,B 0,C 180,E1 25238.441,E2 25238.441} C_VEL
LIN {X 0,Y 571.948,Z 368.821,A -85,B 0,C 180,E1 25237.757,E2 25237.757} C_VEL
LIN {X 0,Y 568.441,Z 364.413,A -85,B 0,C 180,E1 25237.11,E2 25237.11} C_VEL
LIN {X 0,Y 564.13,Z 359.423,A -85,B 0,C 180,E1 25236.299,E2 25236.299} C_VEL
LIN {X 0,Y 562.99,Z 357.664,A -85,B 0,C 180,E1 25236.069,E2 25236.069} C_VEL
LIN {X 0,Y 559.903,Z 354.676,A -85,B 0,C 180,E1 25235.479,E2 25235.479} C_VEL
LIN {X 0,Y 558.155,Z 351.619,A -85,B 0,C 180,E1 25235.103,E2 25235.103} C_VEL
LIN {X 0,Y 555.208,Z 349.426,A -85,B 0,C 180,E1 25234.531,E2 25234.531} C_VEL
LIN {X 0,Y 553.688,Z 346.578,A -85,B 0,C 180,E1 25234.186,E2 25234.186} C_VEL
LIN {X 0,Y 553.423,Z 345.286,A -85,B 0,C 180,E1 25234.092,E2 25234.092} C_VEL
LIN {X 0,Y 553.418,Z 345.297,A -85,B 0,C 180,E1 25230.685,E2 25230.685} C_VEL
LIN {X 0,Y 553.443,Z 345.228,A -85,B 0,C 180,E1 25227.666,E2 25227.666} C_VEL
LIN {X 0,Y 553.416,Z 345.294,A -85,B 0,C 180,E1 25224.415,E2 25224.415} C_VEL
LIN {X 0,Y 553.477,Z 345.221,A -85,B 0,C 180,E1 25221.227,E2 25221.227} C_VEL
LIN {X 0,Y 553.415,Z 345.295,A -85,B 0,C 180,E1 25217.996,E2 25217.996} C_VEL
LIN {X 0,Y 553.467,Z 345.288,A -85,B 0,C 180,E1 25214.758,E2 25214.758} C_VEL
LIN {X 0,Y 553.418,Z 345.293,A -85,B 0,C 180,E1 25211.675,E2 25211.675} C_VEL
LIN {X 0,Y 553.438,Z 345.293,A -85,B 0,C 180,E1 25208.31,E2 25208.31} C_VEL
LIN {X 0,Y 553.426,Z 345.282,A -85,B 0,C 180,E1 25205.391,E2 25205.391} C_VEL
LIN {X 0,Y 553.425,Z 345.282,A -85,B 0,C 180,E1 25201.967,E2 25201.967} C_VEL
LIN {X 0,Y 553.438,Z 345.276,A -85,B 0,C 180,E1 25199.068,E2 25199.068} C_VEL
LIN {X 0,Y 553.423,Z 345.276,A -85,B 0,C 180,E1 25195.752,E2 25195.752} C_VEL
LIN {X 0,Y 553.468,Z 345.277,A -85,B 0,C 180,E1 25192.63,E2 25192.63} C_VEL
LIN {X 0,Y 553.419,Z 345.279,A -85,B 0,C 180,E1 25189.369,E2 25189.369} C_VEL
LIN {X 0,Y 553.481,Z 345.228,A -85,B 0,C 180,E1 25186.097,E2 25186.097} C_VEL
LIN {X 0,Y 553.423,Z 345.276,A -85,B 0,C 180,E1 25182.981,E2 25182.981} C_VEL
LIN {X 0,Y 553.45,Z 345.241,A -85,B 0,C 180,E1 25179.655,E2 25179.655} C_VEL
LIN {X 0,Y 553.421,Z 345.26,A -85,B 0,C 180,E1 25176.804,E2 25176.804} C_VEL
LIN {X 0,Y 553.456,Z 345.257,A -85,B 0,C 180,E1 25173.497,E2 25173.497} C_VEL
LIN {X 0,Y 553.473,Z 345.5,A -85,B 0,C 180,E1 25173.325,E2 25173.325} C_VEL
LIN {X 0,Y 554.984,Z 349.121,A -85,B 0,C 180,E1 25172.621,E2 25172.621} C_VEL
LIN {X 0,Y 557.349,Z 351.748,A -85,B 0,C 180,E1 25172.138,E2 25172.138} C_VEL
LIN {X 0,Y 560.636,Z 355.727,A -85,B 0,C 180,E1 25171.476,E2 25171.476} C_VEL
LIN {X 0,Y 565.004,Z 361.353,A -85,B 0,C 180,E1 25170.617,E2 25170.617} C_VEL
LIN {X 0,Y 577.474,Z 377.449,A -85,B 0,C 180,E1 25168.327,E2 25168.327} C_VEL
LIN {X 0,Y 592.499,Z 398.074,A -85,B 0,C 180,E1 25165.808,E2 25165.808} C_VEL
LIN {X 0,Y 609.107,Z 421.578,A -85,B 0,C 180,E1 25163.277,E2 25163.277} C_VEL
LIN {X 0,Y 614.057,Z 429.263,A -85,B 0,C 180,E1 25162.555,E2 25162.555} C_VEL
LIN {X 0,Y 607.504,Z 635.821,A -85,B 0,C 180,E1 25159.58,E2 25159.58} C_VEL
LIN {X 0,Y 601.502,Z 826.154,A -85,B 0,C 180,E1 25156.864,E2 25156.864} C_VEL
LIN {X 0,Y 600.041,Z 849.804,A -85,B 0,C 180,E1 25156.434,E2 25156.434} C_VEL
LIN {X 0,Y 597.608,Z 878.701,A -85,B 0,C 180,E1 25155.719,E2 25155.719} C_VEL
LIN {X 0,Y 595.334,Z 900.583,A -85,B 0,C 180,E1 25155.03,E2 25155.03} C_VEL
LIN {X 0,Y 592.95,Z 920.802,A -85,B 0,C 180,E1 25154.275,E2 25154.275} C_VEL
LIN {X 0,Y 590.453,Z 940.172,A -85,B 0,C 180,E1 25153.433,E2 25153.433} C_VEL
LIN {X 0,Y 587.705,Z 959.352,A -85,B 0,C 180,E1 25152.486,E2 25152.486} C_VEL
LIN {X 0,Y 584.549,Z 980.083,A -85,B 0,C 180,E1 25151.318,E2 25151.318} C_VEL
LIN {X 0,Y 580.379,Z 1005.82,A -85,B 0,C 180,E1 25149.637,E2 25149.637} C_VEL
LIN {X 0,Y 577.102,Z 1024.842,A -85,B 0,C 180,E1 25148.208,E2 25148.208} C_VEL
LIN {X 0,Y 574.032,Z 1042.219,A -85,B 0,C 180,E1 25146.749,E2 25146.749} C_VEL
LIN {X 0,Y 571.11,Z 1058.494,A -85,B 0,C 180,E1 25145.23,E2 25145.23} C_VEL
LIN {X 0,Y 568.193,Z 1074.819,A -85,B 0,C 180,E1 25143.542,E2 25143.542} C_VEL
LIN {X 0,Y 564.877,Z 1093.745,A -85,B 0,C 180,E1 25141.358,E2 25141.358} C_VEL
LIN {X 0,Y 561.877,Z 1111.065,A -85,B 0,C 180,E1 25139.065,E2 25139.065} C_VEL
LIN {X 0,Y 559.756,Z 1124.376,A -85,B 0,C 180,E1 25137.096,E2 25137.096} C_VEL
LIN {X 0,Y 557.748,Z 1137.631,A -85,B 0,C 180,E1 25134.915,E2 25134.915} C_VEL
LIN {X 0,Y 555.8,Z 1152.163,A -85,B 0,C 180,E1 25132.196,E2 25132.196} C_VEL
LIN {X 0,Y 554.442,Z 1163.606,A -85,B 0,C 180,E1 25129.708,E2 25129.708} C_VEL
LIN {X 0,Y 553.52,Z 1172.704,A -85,B 0,C 180,E1 25127.449,E2 25127.449} C_VEL
LIN {X 0,Y 552.864,Z 1180.922,A -85,B 0,C 180,E1 25125.095,E2 25125.095} C_VEL
LIN {X 0,Y 552.34,Z 1189.025,A -85,B 0,C 180,E1 25122.334,E2 25122.334} C_VEL
LIN {X 0,Y 552.078,Z 1195.294,A -85,B 0,C 180,E1 25119.591,E2 25119.591} C_VEL
LIN {X 0,Y 551.97,Z 1199.532,A -85,B 0,C 180,E1 25117.18,E2 25117.18} C_VEL
LIN {X 0,Y 551.917,Z 1202.669,A -85,B 0,C 180,E1 25114.676,E2 25114.676} C_VEL
LIN {X 0,Y 551.91,Z 1204.6,A -85,B 0,C 180,E1 25111.869,E2 25111.869} C_VEL
LIN {X 0,Y 551.895,Z 1204.872,A -85,B 0,C 180,E1 25109.377,E2 25109.377} C_VEL
LIN {X 0,Y 551.916,Z 1203.978,A -85,B 0,C 180,E1 25106.988,E2 25106.988} C_VEL
LIN {X 0,Y 551.93,Z 1201.872,A -85,B 0,C 180,E1 25104.595,E2 25104.595} C_VEL
LIN {X 0,Y 552,Z 1198.251,A -85,B 0,C 180,E1 25101.983,E2 25101.983} C_VEL
LIN {X 0,Y 552.17,Z 1192.608,A -85,B 0,C 180,E1 25099.145,E2 25099.145} C_VEL
LIN {X 0,Y 552.519,Z 1186.072,A -85,B 0,C 180,E1 25096.607,E2 25096.607} C_VEL
LIN {X 0,Y 552.999,Z 1178.8,A -85,B 0,C 180,E1 25094.264,E2 25094.264} C_VEL
LIN {X 0,Y 553.836,Z 1169.631,A -85,B 0,C 180,E1 25091.739,E2 25091.739} C_VEL
LIN {X 0,Y 555.152,Z 1157.326,A -85,B 0,C 180,E1 25088.887,E2 25088.887} C_VEL
LIN {X 0,Y 556.58,Z 1145.997,A -85,B 0,C 180,E1 25086.609,E2 25086.609} C_VEL
LIN {X 0,Y 558.321,Z 1133.823,A -85,B 0,C 180,E1 25084.432,E2 25084.432} C_VEL
LIN {X 0,Y 560.9,Z 1117.228,A -85,B 0,C 180,E1 25081.811,E2 25081.811} C_VEL
LIN {X 0,Y 563.604,Z 1100.917,A -85,B 0,C 180,E1 25079.567,E2 25079.567} C_VEL
LIN {X 0,Y 566.273,Z 1085.443,A -85,B 0,C 180,E1 25077.656,E2 25077.656} C_VEL
LIN {X 0,Y 569.654,Z 1066.711,A -85,B 0,C 180,E1 25075.586,E2 25075.586} C_VEL
LIN {X 0,Y 573.385,Z 1045.863,A -85,B 0,C 180,E1 25073.576,E2 25073.576} C_VEL
LIN {X 0,Y 576.465,Z 1028.462,A -85,B 0,C 180,E1 25072.084,E2 25072.084} C_VEL
LIN {X 0,Y 579.527,Z 1010.647,A -85,B 0,C 180,E1 25070.715,E2 25070.715} C_VEL
LIN {X 0,Y 582.645,Z 991.957,A -85,B 0,C 180,E1 25069.429,E2 25069.429} C_VEL
LIN {X 0,Y 586.14,Z 970.108,A -85,B 0,C 180,E1 25068.1,E2 25068.1} C_VEL
LIN {X 0,Y 589.842,Z 944.659,A -85,B 0,C 180,E1 25066.778,E2 25066.778} C_VEL
LIN {X 0,Y 592.621,Z 923.312,A -85,B 0,C 180,E1 25065.829,E2 25065.829} C_VEL
LIN {X 0,Y 595.076,Z 902.725,A -85,B 0,C 180,E1 25065.047,E2 25065.047} C_VEL
LIN {X 0,Y 597.271,Z 881.76,A -85,B 0,C 180,E1 25064.372,E2 25064.372} C_VEL
LIN {X 0,Y 599.361,Z 858.427,A -85,B 0,C 180,E1 25063.757,E2 25063.757} C_VEL
LIN {X 0,Y 601.348,Z 829.11,A -85,B 0,C 180,E1 25063.183,E2 25063.183} C_VEL
LIN {X 0,Y 603.548,Z 764.069,A -85,B 0,C 180,E1 25062.243,E2 25062.243} C_VEL
LIN {X 0,Y 610.748,Z 544.807,A -85,B 0,C 180,E1 25059.086,E2 25059.086} C_VEL
LIN {X 0,Y 614.773,Z 428.922,A -85,B 0,C 180,E1 25057.365,E2 25057.365} C_VEL
LIN {X 0,Y 604.714,Z 412.925,A -85,B 0,C 180,E1 25055.681,E2 25055.681} C_VEL
LIN {X 0,Y 594.559,Z 398.254,A -85,B 0,C 180,E1 25053.854,E2 25053.854} C_VEL
LIN {X 0,Y 584.17,Z 384.234,A -85,B 0,C 180,E1 25051.816,E2 25051.816} C_VEL
LIN {X 0,Y 575.747,Z 373.586,A -85,B 0,C 180,E1 25050.011,E2 25050.011} C_VEL
LIN {X 0,Y 571.746,Z 368.482,A -85,B 0,C 180,E1 25049.09,E2 25049.09} C_VEL
LIN {X 0,Y 568.051,Z 364.001,A -85,B 0,C 180,E1 25048.204,E2 25048.204} C_VEL
LIN {X 0,Y 566.73,Z 362.32,A -85,B 0,C 180,E1 25047.875,E2 25047.875} C_VEL
LIN {X 0,Y 563.118,Z 358.059,A -85,B 0,C 180,E1 25046.954,E2 25046.954} C_VEL
LIN {X 0,Y 560.666,Z 355.327,A -85,B 0,C 180,E1 25046.307,E2 25046.307} C_VEL
LIN {X 0,Y 557.208,Z 351.109,A -85,B 0,C 180,E1 25045.34,E2 25045.34} C_VEL
LIN {X 0,Y 554.65,Z 348.613,A -85,B 0,C 180,E1 25044.61,E2 25044.61} C_VEL
LIN {X 0,Y 553.485,Z 345.255,A -85,B 0,C 180,E1 25043.757,E2 25043.757} C_VEL
LIN {X 0,Y 553.442,Z 345.272,A -85,B 0,C 180,E1 25040.628,E2 25040.628} C_VEL
LIN {X 0,Y 553.449,Z 345.239,A -85,B 0,C 180,E1 25037.235,E2 25037.235} C_VEL
LIN {X 0,Y 553.458,Z 345.279,A -85,B 0,C 180,E1 25034.223,E2 25034.223} C_VEL
LIN {X 0,Y 553.44,Z 345.256,A -85,B 0,C 180,E1 25030.83,E2 25030.83} C_VEL
LIN {X 0,Y 553.494,Z 345.24,A -85,B 0,C 180,E1 25027.682,E2 25027.682} C_VEL
LIN {X 0,Y 553.441,Z 345.287,A -85,B 0,C 180,E1 25024.456,E2 25024.456} C_VEL
LIN {X 0,Y 553.499,Z 345.231,A -85,B 0,C 180,E1 25021.242,E2 25021.242} C_VEL
LIN {X 0,Y 553.444,Z 345.291,A -85,B 0,C 180,E1 25018.136,E2 25018.136} C_VEL
LIN {X 0,Y 553.477,Z 345.241,A -85,B 0,C 180,E1 25014.817,E2 25014.817} C_VEL
LIN {X 0,Y 553.446,Z 345.258,A -85,B 0,C 180,E1 25011.794,E2 25011.794} C_VEL
LIN {X 0,Y 553.457,Z 345.282,A -85,B 0,C 180,E1 25008.326,E2 25008.326} C_VEL
LIN {X 0,Y 553.491,Z 345.234,A -85,B 0,C 180,E1 25005.117,E2 25005.117} C_VEL
LIN {X 0,Y 553.52,Z 345.451,A -85,B 0,C 180,E1 25002.589,E2 25002.589} C_VEL
LIN {X 0,Y 554.432,Z 348.204,A -85,B 0,C 180,E1 25002.255,E2 25002.255} C_VEL
LIN {X 0,Y 556.768,Z 350.798,A -85,B 0,C 180,E1 25001.574,E2 25001.574} C_VEL
LIN {X 0,Y 559.174,Z 352.222,A -85,B 0,C 180,E1 25000.94,E2 25000.94} C_VEL
LIN {X 0,Y 561.111,Z 355.711,A -85,B 0,C 180,E1 25000.372,E2 25000.372} C_VEL
LIN {X 0,Y 564.3,Z 358.258,A -85,B 0,C 180,E1 24999.57,E2 24999.57} C_VEL
LIN {X 0,Y 567.778,Z 363.064,A -85,B 0,C 180,E1 24998.675,E2 24998.675} C_VEL
LIN {X 0,Y 570.159,Z 365.142,A -85,B 0,C 180,E1 24998.12,E2 24998.12} C_VEL
LIN {X 0,Y 573.27,Z 369.226,A -85,B 0,C 180,E1 24997.381,E2 24997.381} C_VEL
LIN {X 0,Y 575.321,Z 371.302,A -85,B 0,C 180,E1 24996.926,E2 24996.926} C_VEL
LIN {X 0,Y 578.801,Z 375.655,A -85,B 0,C 180,E1 24996.156,E2 24996.156} C_VEL
LIN {X 0,Y 580.495,Z 377.558,A -85,B 0,C 180,E1 24995.798,E2 24995.798} C_VEL
LIN {X 0,Y 588.506,Z 387.55,A -85,B 0,C 180,E1 24994.164,E2 24994.164} C_VEL
LIN {X 0,Y 598.755,Z 401.409,A -85,B 0,C 180,E1 24992.23,E2 24992.23} C_VEL
LIN {X 0,Y 608.058,Z 415.131,A -85,B 0,C 180,E1 24990.603,E2 24990.603} C_VEL
LIN {X 0,Y 614.812,Z 426.034,A -85,B 0,C 180,E1 24989.484,E2 24989.484} C_VEL
LIN {X 0,Y 607.345,Z 639.327,A -85,B 0,C 180,E1 24986.364,E2 24986.364} C_VEL
LIN {X 0,Y 601.606,Z 816.058,A -85,B 0,C 180,E1 24983.829,E2 24983.829} C_VEL
LIN {X 0,Y 600.526,Z 823.734,A -85,B 0,C 180,E1 24983.785,E2 24983.785} C_VEL
LIN {X 0,Y 594.857,Z 844.253,A -85,B 0,C 180,E1 24983.822,E2 24983.822} C_VEL
LIN {X 0,Y 593.797,Z 850.65,A -85,B 0,C 180,E1 24983.722,E2 24983.722} C_VEL
LIN {X 0,Y 591.696,Z 873.079,A -85,B 0,C 180,E1 24983.123,E2 24983.123} C_VEL
LIN {X 0,Y 589.392,Z 894.225,A -85,B 0,C 180,E1 24982.434,E2 24982.434} C_VEL
LIN {X 0,Y 586.649,Z 916.193,A -85,B 0,C 180,E1 24981.585,E2 24981.585} C_VEL
LIN {X 0,Y 582.933,Z 942.585,A -85,B 0,C 180,E1 24980.366,E2 24980.366} C_VEL
LIN {X 0,Y 579.146,Z 966.451,A -85,B 0,C 180,E1 24979.053,E2 24979.053} C_VEL
LIN {X 0,Y 575.01,Z 990.721,A -85,B 0,C 180,E1 24977.499,E2 24977.499} C_VEL
LIN {X 0,Y 570.899,Z 1013.434,A -85,B 0,C 180,E1 24975.807,E2 24975.807} C_VEL
LIN {X 0,Y 566.605,Z 1036.484,A -85,B 0,C 180,E1 24973.831,E2 24973.831} C_VEL
LIN {X 0,Y 562.917,Z 1055.691,A -85,B 0,C 180,E1 24971.948,E2 24971.948} C_VEL
LIN {X 0,Y 559.638,Z 1073.182,A -85,B 0,C 180,E1 24970.029,E2 24970.029} C_VEL
LIN {X 0,Y 556.024,Z 1092.953,A -85,B 0,C 180,E1 24967.56,E2 24967.56} C_VEL
LIN {X 0,Y 553.349,Z 1108.086,A -85,B 0,C 180,E1 24965.417,E2 24965.417} C_VEL
LIN {X 0,Y 550.859,Z 1123.364,A -85,B 0,C 180,E1 24962.992,E2 24962.992} C_VEL
LIN {X 0,Y 548.659,Z 1137.95,A -85,B 0,C 180,E1 24960.318,E2 24960.318} C_VEL
LIN {X 0,Y 547.121,Z 1149.547,A -85,B 0,C 180,E1 24957.894,E2 24957.894} C_VEL
LIN {X 0,Y 545.801,Z 1161.386,A -85,B 0,C 180,E1 24955.035,E2 24955.035} C_VEL
LIN {X 0,Y 544.972,Z 1170.416,A -85,B 0,C 180,E1 24952.434,E2 24952.434} C_VEL
LIN {X 0,Y 544.459,Z 1177.648,A -85,B 0,C 180,E1 24949.973,E2 24949.973} C_VEL
LIN {X 0,Y 544.134,Z 1184.301,A -85,B 0,C 180,E1 24947.208,E2 24947.208} C_VEL
LIN {X 0,Y 543.984,Z 1189.188,A -85,B 0,C 180,E1 24944.476,E2 24944.476} C_VEL
LIN {X 0,Y 543.927,Z 1192.291,A -85,B 0,C 180,E1 24942.048,E2 24942.048} C_VEL
LIN {X 0,Y 543.911,Z 1194.284,A -85,B 0,C 180,E1 24939.523,E2 24939.523} C_VEL
LIN {X 0,Y 543.905,Z 1194.942,A -85,B 0,C 180,E1 24936.65,E2 24936.65} C_VEL
LIN {X 0,Y 543.91,Z 1194.112,A -85,B 0,C 180,E1 24934.111,E2 24934.111} C_VEL
LIN {X 0,Y 543.923,Z 1192.108,A -85,B 0,C 180,E1 24931.685,E2 24931.685} C_VEL
LIN {X 0,Y 543.988,Z 1188.784,A -85,B 0,C 180,E1 24929.158,E2 24929.158} C_VEL
LIN {X 0,Y 544.154,Z 1183.439,A -85,B 0,C 180,E1 24926.313,E2 24926.313} C_VEL
LIN {X 0,Y 544.486,Z 1177.219,A -85,B 0,C 180,E1 24923.78,E2 24923.78} C_VEL
LIN {X 0,Y 544.991,Z 1170.012,A -85,B 0,C 180,E1 24921.348,E2 24921.348} C_VEL
LIN {X 0,Y 545.925,Z 1160.317,A -85,B 0,C 180,E1 24918.592,E2 24918.592} C_VEL
LIN {X 0,Y 547.156,Z 1149.171,A -85,B 0,C 180,E1 24915.934,E2 24915.934} C_VEL
LIN {X 0,Y 548.721,Z 1137.411,A -85,B 0,C 180,E1 24913.486,E2 24913.486} C_VEL
LIN {X 0,Y 551.023,Z 1122.139,A -85,B 0,C 180,E1 24910.716,E2 24910.716} C_VEL
LIN {X 0,Y 553.489,Z 1107.301,A -85,B 0,C 180,E1 24908.376,E2 24908.376} C_VEL
LIN {X 0,Y 556.425,Z 1090.684,A -85,B 0,C 180,E1 24906.04,E2 24906.04} C_VEL
LIN {X 0,Y 559.953,Z 1071.502,A -85,B 0,C 180,E1 24903.69,E2 24903.69} C_VEL
LIN {X 0,Y 563.093,Z 1054.832,A -85,B 0,C 180,E1 24901.874,E2 24901.874} C_VEL
LIN {X 0,Y 567.012,Z 1034.462,A -85,B 0,C 180,E1 24899.889,E2 24899.889} C_VEL
LIN {X 0,Y 571.082,Z 1012.384,A -85,B 0,C 180,E1 24898.02,E2 24898.02} C_VEL
LIN {X 0,Y 575.23,Z 989.497,A -85,B 0,C 180,E1 24896.325,E2 24896.325} C_VEL
LIN {X 0,Y 579.462,Z 964.583,A -85,B 0,C 180,E1 24894.748,E2 24894.748} C_VEL
LIN {X 0,Y 583.421,Z 939.441,A -85,B 0,C 180,E1 24893.388,E2 24893.388} C_VEL
LIN {X 0,Y 586.931,Z 913.894,A -85,B 0,C 180,E1 24892.23,E2 24892.23} C_VEL
LIN {X 0,Y 589.67,Z 891.849,A -85,B 0,C 180,E1 24891.392,E2 24891.392} C_VEL
LIN {X 0,Y 592.32,Z 867.303,A -85,B 0,C 180,E1 24890.618,E2 24890.618} C_VEL
LIN {X 0,Y 594.679,Z 839.296,A -85,B 0,C 180,E1 24889.937,E2 24889.937} C_VEL
LIN {X 0,Y 596.116,Z 816.583,A -85,B 0,C 180,E1 24889.526,E2 24889.526} C_VEL
LIN {X 0,Y 602.405,Z 624.667,A -85,B 0,C 180,E1 24886.773,E2 24886.773} C_VEL
LIN {X 0,Y 608.841,Z 429.804,A -85,B 0,C 180,E1 24883.951,E2 24883.951} C_VEL
LIN {X 0,Y 596.018,Z 411.343,A -85,B 0,C 180,E1 24882.019,E2 24882.019} C_VEL
LIN {X 0,Y 580.561,Z 390.164,A -85,B 0,C 180,E1 24879.498,E2 24879.498} C_VEL
LIN {X 0,Y 572.382,Z 379.913,A -85,B 0,C 180,E1 24878.072,E2 24878.072} C_VEL
LIN {X 0,Y 568.839,Z 375.506,A -85,B 0,C 180,E1 24877.427,E2 24877.427} C_VEL
LIN {X 0,Y 564.283,Z 369.889,A -85,B 0,C 180,E1 24876.572,E2 24876.572} C_VEL
LIN {X 0,Y 560.77,Z 365.474,A -85,B 0,C 180,E1 24875.887,E2 24875.887} C_VEL
LIN {X 0,Y 556.593,Z 360.769,A -85,B 0,C 180,E1 24875.059,E2 24875.059} C_VEL
LIN {X 0,Y 555.391,Z 358.829,A -85,B 0,C 180,E1 24874.8,E2 24874.8} C_VEL
LIN {X 0,Y 552.246,Z 356.009,A -85,B 0,C 180,E1 24874.167,E2 24874.167} C_VEL
LIN {X 0,Y 550.281,Z 352.627,A -85,B 0,C 180,E1 24873.719,E2 24873.719} C_VEL
LIN {X 0,Y 547.231,Z 350.332,A -85,B 0,C 180,E1 24873.084,E2 24873.084} C_VEL
LIN {X 0,Y 545.694,Z 347.386,A -85,B 0,C 180,E1 24872.709,E2 24872.709} C_VEL
LIN {X 0,Y 545.473,Z 346.276,A -85,B 0,C 180,E1 24872.611,E2 24872.611} C_VEL
LIN {X 0,Y 545.544,Z 346.236,A -85,B 0,C 180,E1 24869.42,E2 24869.42} C_VEL
LIN {X 0,Y 545.47,Z 346.245,A -85,B 0,C 180,E1 24866.217,E2 24866.217} C_VEL
LIN {X 0,Y 545.52,Z 346.226,A -85,B 0,C 180,E1 24862.98,E2 24862.98} C_VEL
LIN {X 0,Y 545.475,Z 346.245,A -85,B 0,C 180,E1 24859.893,E2 24859.893} C_VEL
LIN {X 0,Y 545.494,Z 346.266,A -85,B 0,C 180,E1 24856.506,E2 24856.506} C_VEL
LIN {X 0,Y 545.486,Z 346.268,A -85,B 0,C 180,E1 24853.57,E2 24853.57} C_VEL
LIN {X 0,Y 545.482,Z 346.266,A -85,B 0,C 180,E1 24850.135,E2 24850.135} C_VEL
LIN {X 0,Y 545.535,Z 346.265,A -85,B 0,C 180,E1 24846.948,E2 24846.948} C_VEL
LIN {X 0,Y 545.48,Z 346.279,A -85,B 0,C 180,E1 24843.678,E2 24843.678} C_VEL
LIN {X 0,Y 545.538,Z 346.274,A -85,B 0,C 180,E1 24840.42,E2 24840.42} C_VEL
LIN {X 0,Y 545.486,Z 346.283,A -85,B 0,C 180,E1 24837.268,E2 24837.268} C_VEL
LIN {X 0,Y 545.493,Z 346.282,A -85,B 0,C 180,E1 24833.791,E2 24833.791} C_VEL
LIN {X 0,Y 545.504,Z 346.277,A -85,B 0,C 180,E1 24830.824,E2 24830.824} C_VEL
LIN {X 0,Y 545.48,Z 346.215,A -85,B 0,C 180,E1 24827.508,E2 24827.508} C_VEL
LIN {X 0,Y 545.525,Z 346.272,A -85,B 0,C 180,E1 24824.478,E2 24824.478} C_VEL
LIN {X 0,Y 545.479,Z 346.218,A -85,B 0,C 180,E1 24821.179,E2 24821.179} C_VEL
LIN {X 0,Y 545.561,Z 346.276,A -85,B 0,C 180,E1 24817.931,E2 24817.931} C_VEL
LIN {X 0,Y 545.489,Z 346.261,A -85,B 0,C 180,E1 24814.717,E2 24814.717} C_VEL
LIN {X 0,Y 546.415,Z 349.028,A -85,B 0,C 180,E1 24814.211,E2 24814.211} C_VEL
LIN {X 0,Y 548.963,Z 351.858,A -85,B 0,C 180,E1 24813.651,E2 24813.651} C_VEL
LIN {X 0,Y 555.005,Z 359.301,A -85,B 0,C 180,E1 24812.36,E2 24812.36} C_VEL
LIN {X 0,Y 559.054,Z 364.366,A -85,B 0,C 180,E1 24811.533,E2 24811.533} C_VEL
LIN {X 0,Y 563.886,Z 370.541,A -85,B 0,C 180,E1 24810.582,E2 24810.582} C_VEL
LIN {X 0,Y 574.633,Z 384.567,A -85,B 0,C 180,E1 24808.591,E2 24808.591} C_VEL
LIN {X 0,Y 588.79,Z 404.054,A -85,B 0,C 180,E1 24806.18,E2 24806.18} C_VEL
LIN {X 0,Y 605.736,Z 428.267,A -85,B 0,C 180,E1 24803.555,E2 24803.555} C_VEL
LIN {X 0,Y 608.9,Z 433.273,A -85,B 0,C 180,E1 24803.084,E2 24803.084} C_VEL
LIN {X 0,Y 602.05,Z 641.4,A -85,B 0,C 180,E1 24800.074,E2 24800.074} C_VEL
LIN {X 0,Y 596.029,Z 825.96,A -85,B 0,C 180,E1 24797.429,E2 24797.429} C_VEL
LIN {X 0,Y 594.521,Z 849.476,A -85,B 0,C 180,E1 24797.001,E2 24797.001} C_VEL
LIN {X 0,Y 592.008,Z 878.343,A -85,B 0,C 180,E1 24796.287,E2 24796.287} C_VEL
LIN {X 0,Y 589.614,Z 900.449,A -85,B 0,C 180,E1 24795.59,E2 24795.59} C_VEL
LIN {X 0,Y 587.135,Z 920.675,A -85,B 0,C 180,E1 24794.831,E2 24794.831} C_VEL
LIN {X 0,Y 584.522,Z 940.051,A -85,B 0,C 180,E1 24793.986,E2 24793.986} C_VEL
LIN {X 0,Y 581.506,Z 960.243,A -85,B 0,C 180,E1 24792.981,E2 24792.981} C_VEL
LIN {X 0,Y 577.735,Z 984.103,A -85,B 0,C 180,E1 24791.611,E2 24791.611} C_VEL
LIN {X 0,Y 573.649,Z 1007.61,A -85,B 0,C 180,E1 24790.028,E2 24790.028} C_VEL
LIN {X 0,Y 570.313,Z 1026.075,A -85,B 0,C 180,E1 24788.618,E2 24788.618} C_VEL
LIN {X 0,Y 567.165,Z 1043.118,A -85,B 0,C 180,E1 24787.168,E2 24787.168} C_VEL
LIN {X 0,Y 564.041,Z 1059.816,A -85,B 0,C 180,E1 24785.59,E2 24785.59} C_VEL
LIN {X 0,Y 560.404,Z 1079.379,A -85,B 0,C 180,E1 24783.518,E2 24783.518} C_VEL
LIN {X 0,Y 556.884,Z 1097.98,A -85,B 0,C 180,E1 24781.257,E2 24781.257} C_VEL
LIN {X 0,Y 554.273,Z 1112.604,A -85,B 0,C 180,E1 24779.265,E2 24779.265} C_VEL
LIN {X 0,Y 551.95,Z 1126.475,A -85,B 0,C 180,E1 24777.161,E2 24777.161} C_VEL
LIN {X 0,Y 549.443,Z 1142.55,A -85,B 0,C 180,E1 24774.399,E2 24774.399} C_VEL
LIN {X 0,Y 547.731,Z 1154.763,A -85,B 0,C 180,E1 24771.972,E2 24771.972} C_VEL
LIN {X 0,Y 546.476,Z 1164.981,A -85,B 0,C 180,E1 24769.673,E2 24769.673} C_VEL
LIN {X 0,Y 545.459,Z 1174.728,A -85,B 0,C 180,E1 24767.165,E2 24767.165} C_VEL
LIN {X 0,Y 544.667,Z 1184.555,A -85,B 0,C 180,E1 24764.132,E2 24764.132} C_VEL
LIN {X 0,Y 544.27,Z 1191.079,A -85,B 0,C 180,E1 24761.658,E2 24761.658} C_VEL
LIN {X 0,Y 544.059,Z 1196.177,A -85,B 0,C 180,E1 24759.276,E2 24759.276} C_VEL
LIN {X 0,Y 543.954,Z 1200.486,A -85,B 0,C 180,E1 24756.65,E2 24756.65} C_VEL
LIN {X 0,Y 543.912,Z 1203.499,A -85,B 0,C 180,E1 24753.794,E2 24753.794} C_VEL
LIN {X 0,Y 543.913,Z 1204.713,A -85,B 0,C 180,E1 24751.369,E2 24751.369} C_VEL
LIN {X 0,Y 543.903,Z 1204.826,A -85,B 0,C 180,E1 24749.157,E2 24749.157} C_VEL
LIN {X 0,Y 543.917,Z 1203.907,A -85,B 0,C 180,E1 24746.839,E2 24746.839} C_VEL
LIN {X 0,Y 543.934,Z 1201.756,A -85,B 0,C 180,E1 24744.409,E2 24744.409} C_VEL
LIN {X 0,Y 544.013,Z 1197.908,A -85,B 0,C 180,E1 24741.651,E2 24741.651} C_VEL
LIN {X 0,Y 544.2,Z 1192.308,A -85,B 0,C 180,E1 24738.859,E2 24738.859} C_VEL
LIN {X 0,Y 544.568,Z 1186.069,A -85,B 0,C 180,E1 24736.408,E2 24736.408} C_VEL
LIN {X 0,Y 545.056,Z 1179.153,A -85,B 0,C 180,E1 24734.138,E2 24734.138} C_VEL
LIN {X 0,Y 545.869,Z 1170.678,A -85,B 0,C 180,E1 24731.747,E2 24731.747} C_VEL
LIN {X 0,Y 547.27,Z 1158.354,A -85,B 0,C 180,E1 24728.793,E2 24728.793} C_VEL
LIN {X 0,Y 548.838,Z 1146.568,A -85,B 0,C 180,E1 24726.372,E2 24726.372} C_VEL
LIN {X 0,Y 550.666,Z 1134.456,A -85,B 0,C 180,E1 24724.166,E2 24724.166} C_VEL
LIN {X 0,Y 553.263,Z 1118.749,A -85,B 0,C 180,E1 24721.622,E2 24721.622} C_VEL
LIN {X 0,Y 556.284,Z 1101.361,A -85,B 0,C 180,E1 24719.186,E2 24719.186} C_VEL
LIN {X 0,Y 559.018,Z 1086.367,A -85,B 0,C 180,E1 24717.306,E2 24717.306} C_VEL
LIN {X 0,Y 561.952,Z 1070.764,A -85,B 0,C 180,E1 24715.542,E2 24715.542} C_VEL
LIN {X 0,Y 565.768,Z 1050.837,A -85,B 0,C 180,E1 24713.527,E2 24713.527} C_VEL
LIN {X 0,Y 569.634,Z 1029.804,A -85,B 0,C 180,E1 24711.687,E2 24711.687} C_VEL
LIN {X 0,Y 572.846,Z 1012,A -85,B 0,C 180,E1 24710.296,E2 24710.296} C_VEL
LIN {X 0,Y 575.987,Z 994.035,A -85,B 0,C 180,E1 24709.038,E2 24709.038} C_VEL
LIN {X 0,Y 579.093,Z 975.401,A -85,B 0,C 180,E1 24707.873,E2 24707.873} C_VEL
LIN {X 0,Y 582.386,Z 954.435,A -85,B 0,C 180,E1 24706.716,E2 24706.716} C_VEL
LIN {X 0,Y 586.29,Z 927.161,A -85,B 0,C 180,E1 24705.438,E2 24705.438} C_VEL
LIN {X 0,Y 589.089,Z 904.799,A -85,B 0,C 180,E1 24704.566,E2 24704.566} C_VEL
LIN {X 0,Y 591.433,Z 883.516,A -85,B 0,C 180,E1 24703.868,E2 24703.868} C_VEL
LIN {X 0,Y 593.458,Z 862.2,A -85,B 0,C 180,E1 24703.291,E2 24703.291} C_VEL
LIN {X 0,Y 595.323,Z 838.421,A -85,B 0,C 180,E1 24702.782,E2 24702.782} C_VEL
LIN {X 0,Y 596.994,Z 802.086,A -85,B 0,C 180,E1 24702.214,E2 24702.214} C_VEL
LIN {X 0,Y 604.633,Z 578.658,A -85,B 0,C 180,E1 24698.982,E2 24698.982} C_VEL
LIN {X 0,Y 609.995,Z 433.141,A -85,B 0,C 180,E1 24696.822,E2 24696.822} C_VEL
LIN {X 0,Y 601.201,Z 418.992,A -85,B 0,C 180,E1 24695.306,E2 24695.306} C_VEL
LIN {X 0,Y 591.417,Z 404.679,A -85,B 0,C 180,E1 24693.505,E2 24693.505} C_VEL
LIN {X 0,Y 581.379,Z 391.027,A -85,B 0,C 180,E1 24691.494,E2 24691.494} C_VEL
LIN {X 0,Y 573.371,Z 380.746,A -85,B 0,C 180,E1 24689.745,E2 24689.745} C_VEL
LIN {X 0,Y 569.213,Z 375.481,A -85,B 0,C 180,E1 24688.771,E2 24688.771} C_VEL
LIN {X 0,Y 565.402,Z 370.599,A -85,B 0,C 180,E1 24687.832,E2 24687.832} C_VEL
LIN {X 0,Y 560.803,Z 365.08,A -85,B 0,C 180,E1 24686.642,E2 24686.642} C_VEL
LIN {X 0,Y 555.754,Z 358.99,A -85,B 0,C 180,E1 24685.239,E2 24685.239} C_VEL
LIN {X 0,Y 552.711,Z 356.016,A -85,B 0,C 180,E1 24684.36,E2 24684.36} C_VEL
LIN {X 0,Y 550.212,Z 352.562,A -85,B 0,C 180,E1 24683.566,E2 24683.566} C_VEL
LIN {X 0,Y 547.331,Z 350.41,A -85,B 0,C 180,E1 24682.673,E2 24682.673} C_VEL
LIN {X 0,Y 545.795,Z 347.39,A -85,B 0,C 180,E1 24682.035,E2 24682.035} C_VEL
LIN {X 0,Y 545.544,Z 346.227,A -85,B 0,C 180,E1 24681.687,E2 24681.687} C_VEL
LIN {X 0,Y 545.501,Z 346.241,A -85,B 0,C 180,E1 24678.599,E2 24678.599} C_VEL
LIN {X 0,Y 545.517,Z 346.273,A -85,B 0,C 180,E1 24675.195,E2 24675.195} C_VEL
LIN {X 0,Y 545.524,Z 346.222,A -85,B 0,C 180,E1 24672.061,E2 24672.061} C_VEL
LIN {X 0,Y 545.504,Z 346.266,A -85,B 0,C 180,E1 24668.751,E2 24668.751} C_VEL
LIN {X 0,Y 545.557,Z 346.231,A -85,B 0,C 180,E1 24665.574,E2 24665.574} C_VEL
LIN {X 0,Y 545.497,Z 346.237,A -85,B 0,C 180,E1 24662.311,E2 24662.311} C_VEL
LIN {X 0,Y 545.555,Z 346.266,A -85,B 0,C 180,E1 24659.055,E2 24659.055} C_VEL
LIN {X 0,Y 545.51,Z 346.223,A -85,B 0,C 180,E1 24655.795,E2 24655.795} C_VEL
LIN {X 0,Y 545.514,Z 346.265,A -85,B 0,C 180,E1 24652.416,E2 24652.416} C_VEL
LIN {X 0,Y 545.548,Z 346.235,A -85,B 0,C 180,E1 24649.221,E2 24649.221} C_VEL
LIN {X 0,Y 545.501,Z 346.231,A -85,B 0,C 180,E1 24645.998,E2 24645.998} C_VEL
LIN {X 0,Y 545.588,Z 346.403,A -85,B 0,C 180,E1 24644.793,E2 24644.793} C_VEL
LIN {X 0,Y 546.537,Z 349.241,A -85,B 0,C 180,E1 24644.399,E2 24644.399} C_VEL
LIN {X 0,Y 548.799,Z 351.781,A -85,B 0,C 180,E1 24643.651,E2 24643.651} C_VEL
LIN {X 0,Y 551.374,Z 353.215,A -85,B 0,C 180,E1 24642.888,E2 24642.888} C_VEL
LIN {X 0,Y 553.167,Z 356.608,A -85,B 0,C 180,E1 24642.294,E2 24642.294} C_VEL
LIN {X 0,Y 556.179,Z 359.121,A -85,B 0,C 180,E1 24641.445,E2 24641.445} C_VEL
LIN {X 0,Y 557.148,Z 359.945,A -85,B 0,C 180,E1 24641.18,E2 24641.18} C_VEL
LIN {X 0,Y 559.584,Z 363.649,A -85,B 0,C 180,E1 24640.48,E2 24640.48} C_VEL
LIN {X 0,Y 562.644,Z 366.293,A -85,B 0,C 180,E1 24639.697,E2 24639.697} C_VEL
LIN {X 0,Y 565.646,Z 370.398,A -85,B 0,C 180,E1 24638.916,E2 24638.916} C_VEL
LIN {X 0,Y 567.985,Z 372.61,A -85,B 0,C 180,E1 24638.358,E2 24638.358} C_VEL
LIN {X 0,Y 571.487,Z 376.942,A -85,B 0,C 180,E1 24637.524,E2 24637.524} C_VEL
LIN {X 0,Y 573.096,Z 378.758,A -85,B 0,C 180,E1 24637.157,E2 24637.157} C_VEL
LIN {X 0,Y 576.984,Z 383.375,A -85,B 0,C 180,E1 24636.294,E2 24636.294} C_VEL
LIN {X 0,Y 585.621,Z 394.229,A -85,B 0,C 180,E1 24634.488,E2 24634.488} C_VEL
LIN {X 0,Y 595.742,Z 408.098,A -85,B 0,C 180,E1 24632.539,E2 24632.539} C_VEL
LIN {X 0,Y 604.697,Z 421.457,A -85,B 0,C 180,E1 24630.94,E2 24630.94} C_VEL
LIN {X 0,Y 609.993,Z 430.098,A -85,B 0,C 180,E1 24630.037,E2 24630.037} C_VEL
LIN {X 0,Y 602.06,Z 645.355,A -85,B 0,C 180,E1 24626.867,E2 24626.867} C_VEL
LIN {X 0,Y 596.074,Z 818.046,A -85,B 0,C 180,E1 24624.363,E2 24624.363} C_VEL
LIN {X 0,Y 594.412,Z 843.688,A -85,B 0,C 180,E1 24623.884,E2 24623.884} C_VEL
LIN {X 0,Y 593.797,Z 850.65,A -85,B 0,C 180,E1 24623.722,E2 24623.722} C_VEL
LIN {X 0,Y 592.428,Z 858.204,A -85,B 0,C 180,E1 24623.608,E2 24623.608} C_VEL
LIN {X 0,Y 586.205,Z 878.446,A -85,B 0,C 180,E1 24623.486,E2 24623.486} C_VEL
LIN {X 0,Y 584.949,Z 884.781,A -85,B 0,C 180,E1 24623.336,E2 24623.336} C_VEL
LIN {X 0,Y 581.734,Z 909.987,A -85,B 0,C 180,E1 24622.405,E2 24622.405} C_VEL
LIN {X 0,Y 578.783,Z 930.825,A -85,B 0,C 180,E1 24621.496,E2 24621.496} C_VEL
LIN {X 0,Y 575.431,Z 952.366,A -85,B 0,C 180,E1 24620.409,E2 24620.409} C_VEL
LIN {X 0,Y 571.136,Z 977.785,A -85,B 0,C 180,E1 24618.908,E2 24618.908} C_VEL
LIN {X 0,Y 567.076,Z 999.886,A -85,B 0,C 180,E1 24617.384,E2 24617.384} C_VEL
LIN {X 0,Y 562.656,Z 1022.904,A -85,B 0,C 180,E1 24615.559,E2 24615.559} C_VEL
LIN {X 0,Y 558.519,Z 1043.582,A -85,B 0,C 180,E1 24613.675,E2 24613.675} C_VEL
LIN {X 0,Y 554.44,Z 1064.108,A -85,B 0,C 180,E1 24611.546,E2 24611.546} C_VEL
LIN {X 0,Y 550.908,Z 1081.938,A -85,B 0,C 180,E1 24609.437,E2 24609.437} C_VEL
LIN {X 0,Y 547.985,Z 1097.245,A -85,B 0,C 180,E1 24607.416,E2 24607.416} C_VEL
LIN {X 0,Y 544.903,Z 1114.253,A -85,B 0,C 180,E1 24604.891,E2 24604.891} C_VEL
LIN {X 0,Y 542.425,Z 1128.783,A -85,B 0,C 180,E1 24602.406,E2 24602.406} C_VEL
LIN {X 0,Y 540.478,Z 1141.438,A -85,B 0,C 180,E1 24599.966,E2 24599.966} C_VEL
LIN {X 0,Y 538.708,Z 1154.679,A -85,B 0,C 180,E1 24597.01,E2 24597.01} C_VEL
LIN {X 0,Y 537.618,Z 1164.263,A -85,B 0,C 180,E1 24594.502,E2 24594.502} C_VEL
LIN {X 0,Y 536.838,Z 1173.263,A -85,B 0,C 180,E1 24591.755,E2 24591.755} C_VEL
LIN {X 0,Y 536.309,Z 1181.031,A -85,B 0,C 180,E1 24588.816,E2 24588.816} C_VEL
LIN {X 0,Y 536.075,Z 1186.195,A -85,B 0,C 180,E1 24586.358,E2 24586.358} C_VEL
LIN {X 0,Y 535.956,Z 1190.3,A -85,B 0,C 180,E1 24583.815,E2 24583.815} C_VEL
LIN {X 0,Y 535.916,Z 1193.397,A -85,B 0,C 180,E1 24580.97,E2 24580.97} C_VEL
LIN {X 0,Y 535.913,Z 1194.714,A -85,B 0,C 180,E1 24578.368,E2 24578.368} C_VEL
LIN {X 0,Y 535.913,Z 1194.831,A -85,B 0,C 180,E1 24576.105,E2 24576.105} C_VEL
LIN {X 0,Y 535.909,Z 1193.908,A -85,B 0,C 180,E1 24573.744,E2 24573.744} C_VEL
LIN {X 0,Y 535.936,Z 1191.662,A -85,B 0,C 180,E1 24571.176,E2 24571.176} C_VEL
LIN {X 0,Y 536.03,Z 1187.564,A -85,B 0,C 180,E1 24568.29,E2 24568.29} C_VEL
LIN {X 0,Y 536.22,Z 1182.46,A -85,B 0,C 180,E1 24565.723,E2 24565.723} C_VEL
LIN {X 0,Y 536.601,Z 1176.348,A -85,B 0,C 180,E1 24563.259,E2 24563.259} C_VEL
LIN {X 0,Y 537.271,Z 1168.162,A -85,B 0,C 180,E1 24560.527,E2 24560.527} C_VEL
LIN {X 0,Y 538.339,Z 1157.751,A -85,B 0,C 180,E1 24557.667,E2 24557.667} C_VEL
LIN {X 0,Y 539.664,Z 1147.238,A -85,B 0,C 180,E1 24555.186,E2 24555.186} C_VEL
LIN {X 0,Y 541.668,Z 1133.578,A -85,B 0,C 180,E1 24552.379,E2 24552.379} C_VEL
LIN {X 0,Y 543.961,Z 1119.542,A -85,B 0,C 180,E1 24549.896,E2 24549.896} C_VEL
LIN {X 0,Y 546.506,Z 1105.172,A -85,B 0,C 180,E1 24547.633,E2 24547.633} C_VEL
LIN {X 0,Y 550.02,Z 1086.564,A -85,B 0,C 180,E1 24545.055,E2 24545.055} C_VEL
LIN {X 0,Y 553.274,Z 1069.863,A -85,B 0,C 180,E1 24543.025,E2 24543.025} C_VEL
LIN {X 0,Y 556.783,Z 1052.363,A -85,B 0,C 180,E1 24541.114,E2 24541.114} C_VEL
LIN {X 0,Y 561.186,Z 1030.186,A -85,B 0,C 180,E1 24538.984,E2 24538.984} C_VEL
LIN {X 0,Y 565.581,Z 1007.696,A -85,B 0,C 180,E1 24537.114,E2 24537.114} C_VEL
LIN {X 0,Y 569.969,Z 984.171,A -85,B 0,C 180,E1 24535.425,E2 24535.425} C_VEL
LIN {X 0,Y 573.865,Z 962.031,A -85,B 0,C 180,E1 24534.044,E2 24534.044} C_VEL
LIN {X 0,Y 577.997,Z 936.328,A -85,B 0,C 180,E1 24532.676,E2 24532.676} C_VEL
LIN {X 0,Y 581.164,Z 913.985,A -85,B 0,C 180,E1 24531.668,E2 24531.668} C_VEL
LIN {X 0,Y 583.827,Z 893.445,A -85,B 0,C 180,E1 24530.881,E2 24530.881} C_VEL
LIN {X 0,Y 586.232,Z 872.162,A -85,B 0,C 180,E1 24530.191,E2 24530.191} C_VEL
LIN {X 0,Y 588.551,Z 847.91,A -85,B 0,C 180,E1 24529.552,E2 24529.552} C_VEL
LIN {X 0,Y 590.529,Z 819.657,A -85,B 0,C 180,E1 24529.003,E2 24529.003} C_VEL
LIN {X 0,Y 592.888,Z 754.003,A -85,B 0,C 180,E1 24528.046,E2 24528.046} C_VEL
LIN {X 0,Y 600.355,Z 531.438,A -85,B 0,C 180,E1 24524.841,E2 24524.841} C_VEL
LIN {X 0,Y 603.619,Z 433.601,A -85,B 0,C 180,E1 24523.396,E2 24523.396} C_VEL
LIN {X 0,Y 590.959,Z 415.688,A -85,B 0,C 180,E1 24521.449,E2 24521.449} C_VEL
LIN {X 0,Y 577.719,Z 397.207,A -85,B 0,C 180,E1 24519.242,E2 24519.242} C_VEL
LIN {X 0,Y 566.362,Z 382.799,A -85,B 0,C 180,E1 24517.205,E2 24517.205} C_VEL
LIN {X 0,Y 560.996,Z 376.347,A -85,B 0,C 180,E1 24516.186,E2 24516.186} C_VEL
LIN {X 0,Y 556.939,Z 371.323,A -85,B 0,C 180,E1 24515.38,E2 24515.38} C_VEL
LIN {X 0,Y 553.422,Z 367.016,A -85,B 0,C 180,E1 24514.658,E2 24514.658} C_VEL
LIN {X 0,Y 552.182,Z 365.592,A -85,B 0,C 180,E1 24514.4,E2 24514.4} C_VEL
LIN {X 0,Y 548.947,Z 362.039,A -85,B 0,C 180,E1 24513.717,E2 24513.717} C_VEL
LIN {X 0,Y 547.582,Z 359.846,A -85,B 0,C 180,E1 24513.404,E2 24513.404} C_VEL
LIN {X 0,Y 544.395,Z 356.984,A -85,B 0,C 180,E1 24512.718,E2 24512.718} C_VEL
LIN {X 0,Y 542.478,Z 353.691,A -85,B 0,C 180,E1 24512.249,E2 24512.249} C_VEL
LIN {X 0,Y 539.455,Z 351.469,A -85,B 0,C 180,E1 24511.576,E2 24511.576} C_VEL
LIN {X 0,Y 537.828,Z 348.481,A -85,B 0,C 180,E1 24511.152,E2 24511.152} C_VEL
LIN {X 0,Y 537.567,Z 347.265,A -85,B 0,C 180,E1 24511.058,E2 24511.058} C_VEL
LIN {X 0,Y 537.537,Z 347.204,A -85,B 0,C 180,E1 24507.954,E2 24507.954} C_VEL
LIN {X 0,Y 537.543,Z 347.272,A -85,B 0,C 180,E1 24504.507,E2 24504.507} C_VEL
LIN {X 0,Y 537.593,Z 347.194,A -85,B 0,C 180,E1 24501.266,E2 24501.266} C_VEL
LIN {X 0,Y 537.538,Z 347.273,A -85,B 0,C 180,E1 24497.986,E2 24497.986} C_VEL
LIN {X 0,Y 537.577,Z 347.266,A -85,B 0,C 180,E1 24494.653,E2 24494.653} C_VEL
LIN {X 0,Y 537.552,Z 347.272,A -85,B 0,C 180,E1 24491.48,E2 24491.48} C_VEL
LIN {X 0,Y 537.542,Z 347.272,A -85,B 0,C 180,E1 24488.019,E2 24488.019} C_VEL
LIN {X 0,Y 537.592,Z 347.261,A -85,B 0,C 180,E1 24484.908,E2 24484.908} C_VEL
LIN {X 0,Y 537.539,Z 347.265,A -85,B 0,C 180,E1 24481.599,E2 24481.599} C_VEL
LIN {X 0,Y 537.599,Z 347.251,A -85,B 0,C 180,E1 24478.401,E2 24478.401} C_VEL
LIN {X 0,Y 537.547,Z 347.253,A -85,B 0,C 180,E1 24475.198,E2 24475.198} C_VEL
LIN {X 0,Y 537.552,Z 347.256,A -85,B 0,C 180,E1 24471.701,E2 24471.701} C_VEL
LIN {X 0,Y 537.581,Z 347.217,A -85,B 0,C 180,E1 24468.572,E2 24468.572} C_VEL
LIN {X 0,Y 537.541,Z 347.231,A -85,B 0,C 180,E1 24465.291,E2 24465.291} C_VEL
LIN {X 0,Y 537.608,Z 347.212,A -85,B 0,C 180,E1 24462.129,E2 24462.129} C_VEL
LIN {X 0,Y 537.547,Z 347.243,A -85,B 0,C 180,E1 24458.847,E2 24458.847} C_VEL
LIN {X 0,Y 537.617,Z 347.372,A -85,B 0,C 180,E1 24456.139,E2 24456.139} C_VEL
LIN {X 0,Y 538.073,Z 349.07,A -85,B 0,C 180,E1 24455.884,E2 24455.884} C_VEL
LIN {X 0,Y 539.871,Z 351.901,A -85,B 0,C 180,E1 24455.43,E2 24455.43} C_VEL
LIN {X 0,Y 542.539,Z 354.06,A -85,B 0,C 180,E1 24454.832,E2 24454.832} C_VEL
LIN {X 0,Y 545.845,Z 358.503,A -85,B 0,C 180,E1 24454.065,E2 24454.065} C_VEL
LIN {X 0,Y 547.571,Z 360.392,A -85,B 0,C 180,E1 24453.687,E2 24453.687} C_VEL
LIN {X 0,Y 552.568,Z 366.626,A -85,B 0,C 180,E1 24452.608,E2 24452.608} C_VEL
LIN {X 0,Y 556.471,Z 371.57,A -85,B 0,C 180,E1 24451.799,E2 24451.799} C_VEL
LIN {X 0,Y 561.379,Z 377.906,A -85,B 0,C 180,E1 24450.818,E2 24450.818} C_VEL
LIN {X 0,Y 571.327,Z 390.929,A -85,B 0,C 180,E1 24448.946,E2 24448.946} C_VEL
LIN {X 0,Y 585.608,Z 410.808,A -85,B 0,C 180,E1 24446.471,E2 24446.471} C_VEL
LIN {X 0,Y 602.11,Z 434.547,A -85,B 0,C 180,E1 24443.876,E2 24443.876} C_VEL
LIN {X 0,Y 603.78,Z 437.3,A -85,B 0,C 180,E1 24443.621,E2 24443.621} C_VEL
LIN {X 0,Y 596.607,Z 647.152,A -85,B 0,C 180,E1 24440.573,E2 24440.573} C_VEL
LIN {X 0,Y 590.579,Z 825.927,A -85,B 0,C 180,E1 24437.998,E2 24437.998} C_VEL
LIN {X 0,Y 589.009,Z 849.671,A -85,B 0,C 180,E1 24437.565,E2 24437.565} C_VEL
LIN {X 0,Y 586.404,Z 878.505,A -85,B 0,C 180,E1 24436.849,E2 24436.849} C_VEL
LIN {X 0,Y 583.862,Z 901.057,A -85,B 0,C 180,E1 24436.133,E2 24436.133} C_VEL
LIN {X 0,Y 581.379,Z 920.547,A -85,B 0,C 180,E1 24435.398,E2 24435.398} C_VEL
LIN {X 0,Y 578.647,Z 939.926,A -85,B 0,C 180,E1 24434.55,E2 24434.55} C_VEL
LIN {X 0,Y 575.524,Z 960.023,A -85,B 0,C 180,E1 24433.545,E2 24433.545} C_VEL
LIN {X 0,Y 571.648,Z 983.469,A -85,B 0,C 180,E1 24432.194,E2 24432.194} C_VEL
LIN {X 0,Y 567.437,Z 1006.762,A -85,B 0,C 180,E1 24430.623,E2 24430.623} C_VEL
LIN {X 0,Y 563.958,Z 1025.175,A -85,B 0,C 180,E1 24429.213,E2 24429.213} C_VEL
LIN {X 0,Y 560.57,Z 1042.654,A -85,B 0,C 180,E1 24427.719,E2 24427.719} C_VEL
LIN {X 0,Y 557.268,Z 1059.519,A -85,B 0,C 180,E1 24426.114,E2 24426.114} C_VEL
LIN {X 0,Y 553.705,Z 1077.857,A -85,B 0,C 180,E1 24424.166,E2 24424.166} C_VEL
LIN {X 0,Y 549.9,Z 1097.133,A -85,B 0,C 180,E1 24421.823,E2 24421.823} C_VEL
LIN {X 0,Y 547.09,Z 1111.832,A -85,B 0,C 180,E1 24419.809,E2 24419.809} C_VEL
LIN {X 0,Y 544.704,Z 1125.168,A -85,B 0,C 180,E1 24417.774,E2 24417.774} C_VEL
LIN {X 0,Y 542.306,Z 1139.531,A -85,B 0,C 180,E1 24415.324,E2 24415.324} C_VEL
LIN {X 0,Y 540.146,Z 1153.749,A -85,B 0,C 180,E1 24412.523,E2 24412.523} C_VEL
LIN {X 0,Y 538.779,Z 1164.062,A -85,B 0,C 180,E1 24410.192,E2 24410.192} C_VEL
LIN {X 0,Y 537.746,Z 1173.107,A -85,B 0,C 180,E1 24407.866,E2 24407.866} C_VEL
LIN {X 0,Y 536.938,Z 1181.979,A -85,B 0,C 180,E1 24405.222,E2 24405.222} C_VEL
LIN {X 0,Y 536.35,Z 1190.059,A -85,B 0,C 180,E1 24402.27,E2 24402.27} C_VEL
LIN {X 0,Y 536.098,Z 1195.495,A -85,B 0,C 180,E1 24399.772,E2 24399.772} C_VEL
LIN {X 0,Y 535.98,Z 1199.526,A -85,B 0,C 180,E1 24397.395,E2 24397.395} C_VEL
LIN {X 0,Y 535.924,Z 1202.55,A -85,B 0,C 180,E1 24394.923,E2 24394.923} C_VEL
LIN {X 0,Y 535.911,Z 1204.577,A -85,B 0,C 180,E1 24392.031,E2 24392.031} C_VEL
LIN {X 0,Y 535.895,Z 1204.872,A -85,B 0,C 180,E1 24389.359,E2 24389.359} C_VEL
LIN {X 0,Y 535.915,Z 1204.04,A -85,B 0,C 180,E1 24387.006,E2 24387.006} C_VEL
LIN {X 0,Y 535.931,Z 1202.094,A -85,B 0,C 180,E1 24384.648,E2 24384.648} C_VEL
LIN {X 0,Y 535.984,Z 1199.046,A -85,B 0,C 180,E1 24382.281,E2 24382.281} C_VEL
LIN {X 0,Y 536.153,Z 1194.256,A -85,B 0,C 180,E1 24379.578,E2 24379.578} C_VEL
LIN {X 0,Y 536.548,Z 1187.175,A -85,B 0,C 180,E1 24376.602,E2 24376.602} C_VEL
LIN {X 0,Y 537.085,Z 1179.858,A -85,B 0,C 180,E1 24374.118,E2 24374.118} C_VEL
LIN {X 0,Y 537.886,Z 1171.844,A -85,B 0,C 180,E1 24371.79,E2 24371.79} C_VEL
LIN {X 0,Y 539.073,Z 1161.773,A -85,B 0,C 180,E1 24369.252,E2 24369.252} C_VEL
LIN {X 0,Y 540.935,Z 1148.287,A -85,B 0,C 180,E1 24366.353,E2 24366.353} C_VEL
LIN {X 0,Y 542.817,Z 1136.359,A -85,B 0,C 180,E1 24364.116,E2 24364.116} C_VEL
LIN {X 0,Y 544.999,Z 1123.405,A -85,B 0,C 180,E1 24361.943,E2 24361.943} C_VEL
LIN {X 0,Y 548.028,Z 1107.205,A -85,B 0,C 180,E1 24359.522,E2 24359.522} C_VEL
LIN {X 0,Y 551.436,Z 1089.143,A -85,B 0,C 180,E1 24357.17,E2 24357.17} C_VEL
LIN {X 0,Y 554.456,Z 1073.796,A -85,B 0,C 180,E1 24355.386,E2 24355.386} C_VEL
LIN {X 0,Y 557.688,Z 1057.276,A -85,B 0,C 180,E1 24353.663,E2 24353.663} C_VEL
LIN {X 0,Y 561.303,Z 1038.86,A -85,B 0,C 180,E1 24351.941,E2 24351.941} C_VEL
LIN {X 0,Y 565.926,Z 1014.829,A -85,B 0,C 180,E1 24349.977,E2 24349.977} C_VEL
LIN {X 0,Y 569.418,Z 995.779,A -85,B 0,C 180,E1 24348.616,E2 24348.616} C_VEL
LIN {X 0,Y 572.67,Z 977.168,A -85,B 0,C 180,E1 24347.432,E2 24347.432} C_VEL
LIN {X 0,Y 575.816,Z 958.033,A -85,B 0,C 180,E1 24346.352,E2 24346.352} C_VEL
LIN {X 0,Y 578.964,Z 937.568,A -85,B 0,C 180,E1 24345.342,E2 24345.342} C_VEL
LIN {X 0,Y 582.543,Z 912.073,A -85,B 0,C 180,E1 24344.262,E2 24344.262} C_VEL
LIN {X 0,Y 585.611,Z 885.846,A -85,B 0,C 180,E1 24343.367,E2 24343.367} C_VEL
LIN {X 0,Y 587.795,Z 864.361,A -85,B 0,C 180,E1 24342.771,E2 24342.771} C_VEL
LIN {X 0,Y 589.586,Z 842.958,A -85,B 0,C 180,E1 24342.293,E2 24342.293} C_VEL
LIN {X 0,Y 591.036,Z 819.276,A -85,B 0,C 180,E1 24341.886,E2 24341.886} C_VEL
LIN {X 0,Y 599.063,Z 597.009,A -85,B 0,C 180,E1 24338.643,E2 24338.643} C_VEL
LIN {X 0,Y 605.246,Z 437.159,A -85,B 0,C 180,E1 24336.259,E2 24336.259} C_VEL
LIN {X 0,Y 595.151,Z 421.104,A -85,B 0,C 180,E1 24334.455,E2 24334.455} C_VEL
LIN {X 0,Y 586.173,Z 408.207,A -85,B 0,C 180,E1 24332.734,E2 24332.734} C_VEL
LIN {X 0,Y 577.969,Z 397.034,A -85,B 0,C 180,E1 24331.034,E2 24331.034} C_VEL
LIN {X 0,Y 571.112,Z 388.017,A -85,B 0,C 180,E1 24329.499,E2 24329.499} C_VEL
LIN {X 0,Y 566.702,Z 382.458,A -85,B 0,C 180,E1 24328.45,E2 24328.45} C_VEL
LIN {X 0,Y 562.014,Z 376.534,A -85,B 0,C 180,E1 24327.266,E2 24327.266} C_VEL
LIN {X 0,Y 556.83,Z 370.268,A -85,B 0,C 180,E1 24325.871,E2 24325.871} C_VEL
LIN {X 0,Y 553.261,Z 366.03,A -85,B 0,C 180,E1 24324.847,E2 24324.847} C_VEL
LIN {X 0,Y 550.37,Z 362.76,A -85,B 0,C 180,E1 24323.974,E2 24323.974} C_VEL
LIN {X 0,Y 548.3,Z 360.128,A -85,B 0,C 180,E1 24323.311,E2 24323.311} C_VEL
LIN {X 0,Y 545.332,Z 357.603,A -85,B 0,C 180,E1 24322.362,E2 24322.362} C_VEL
LIN {X 0,Y 543.147,Z 353.869,A -85,B 0,C 180,E1 24321.547,E2 24321.547} C_VEL
LIN {X 0,Y 539.947,Z 352.008,A -85,B 0,C 180,E1 24320.431,E2 24320.431} C_VEL
LIN {X 0,Y 538.072,Z 349.114,A -85,B 0,C 180,E1 24319.655,E2 24319.655} C_VEL
LIN {X 0,Y 537.58,Z 347.248,A -85,B 0,C 180,E1 24319.334,E2 24319.334} C_VEL
LIN {X 0,Y 537.595,Z 347.227,A -85,B 0,C 180,E1 24316.089,E2 24316.089} C_VEL
LIN {X 0,Y 537.557,Z 347.216,A -85,B 0,C 180,E1 24312.788,E2 24312.788} C_VEL
LIN {X 0,Y 537.625,Z 347.264,A -85,B 0,C 180,E1 24309.528,E2 24309.528} C_VEL
LIN {X 0,Y 537.559,Z 347.213,A -85,B 0,C 180,E1 24306.301,E2 24306.301} C_VEL
LIN {X 0,Y 537.582,Z 347.237,A -85,B 0,C 180,E1 24302.879,E2 24302.879} C_VEL
LIN {X 0,Y 537.592,Z 347.232,A -85,B 0,C 180,E1 24299.68,E2 24299.68} C_VEL
LIN {X 0,Y 537.562,Z 347.215,A -85,B 0,C 180,E1 24296.374,E2 24296.374} C_VEL
LIN {X 0,Y 537.636,Z 347.264,A -85,B 0,C 180,E1 24293.057,E2 24293.057} C_VEL
LIN {X 0,Y 537.57,Z 347.217,A -85,B 0,C 180,E1 24289.71,E2 24289.71} C_VEL
LIN {X 0,Y 537.62,Z 347.457,A -85,B 0,C 180,E1 24287.377,E2 24287.377} C_VEL
LIN {X 0,Y 538.592,Z 350.166,A -85,B 0,C 180,E1 24286.909,E2 24286.909} C_VEL
LIN {X 0,Y 540.83,Z 352.725,A -85,B 0,C 180,E1 24286.038,E2 24286.038} C_VEL
LIN {X 0,Y 543.639,Z 354.24,A -85,B 0,C 180,E1 24285.078,E2 24285.078} C_VEL
LIN {X 0,Y 545.37,Z 357.649,A -85,B 0,C 180,E1 24284.419,E2 24284.419} C_VEL
LIN {X 0,Y 548.331,Z 360.165,A -85,B 0,C 180,E1 24283.473,E2 24283.473} C_VEL
LIN {X 0,Y 549.474,Z 360.969,A -85,B 0,C 180,E1 24283.127,E2 24283.127} C_VEL
LIN {X 0,Y 551.764,Z 364.615,A -85,B 0,C 180,E1 24282.384,E2 24282.384} C_VEL
LIN {X 0,Y 555.111,Z 367.43,A -85,B 0,C 180,E1 24281.436,E2 24281.436} C_VEL
LIN {X 0,Y 557.887,Z 371.358,A -85,B 0,C 180,E1 24280.636,E2 24280.636} C_VEL
LIN {X 0,Y 560.545,Z 373.744,A -85,B 0,C 180,E1 24279.944,E2 24279.944} C_VEL
LIN {X 0,Y 563.906,Z 378.105,A -85,B 0,C 180,E1 24279.066,E2 24279.066} C_VEL
LIN {X 0,Y 565.921,Z 380.179,A -85,B 0,C 180,E1 24278.574,E2 24278.574} C_VEL
LIN {X 0,Y 569.709,Z 384.647,A -85,B 0,C 180,E1 24277.668,E2 24277.668} C_VEL
LIN {X 0,Y 574.748,Z 390.707,A -85,B 0,C 180,E1 24276.522,E2 24276.522} C_VEL
LIN {X 0,Y 583.185,Z 401.525,A -85,B 0,C 180,E1 24274.728,E2 24274.728} C_VEL
LIN {X 0,Y 592.862,Z 414.965,A -85,B 0,C 180,E1 24272.83,E2 24272.83} C_VEL
LIN {X 0,Y 601.478,Z 427.972,A -85,B 0,C 180,E1 24271.259,E2 24271.259} C_VEL
LIN {X 0,Y 605.243,Z 434.304,A -85,B 0,C 180,E1 24270.597,E2 24270.597} C_VEL
LIN {X 0,Y 596.936,Z 648.964,A -85,B 0,C 180,E1 24267.416,E2 24267.416} C_VEL
LIN {X 0,Y 590.744,Z 818.126,A -85,B 0,C 180,E1 24264.943,E2 24264.943} C_VEL
LIN {X 0,Y 589.016,Z 843.632,A -85,B 0,C 180,E1 24264.463,E2 24264.463} C_VEL
LIN {X 0,Y 586.422,Z 870.868,A -85,B 0,C 180,E1 24263.763,E2 24263.763} C_VEL
LIN {X 0,Y 584.949,Z 884.781,A -85,B 0,C 180,E1 24263.336,E2 24263.336} C_VEL
LIN {X 0,Y 583.334,Z 892.293,A -85,B 0,C 180,E1 24263.152,E2 24263.152} C_VEL
LIN {X 0,Y 576.648,Z 911.052,A -85,B 0,C 180,E1 24262.874,E2 24262.874} C_VEL
LIN {X 0,Y 574.961,Z 918.119,A -85,B 0,C 180,E1 24262.651,E2 24262.651} C_VEL
LIN {X 0,Y 570.782,Z 944.888,A -85,B 0,C 180,E1 24261.377,E2 24261.377} C_VEL
LIN {X 0,Y 567.211,Z 965.68,A -85,B 0,C 180,E1 24260.215,E2 24260.215} C_VEL
LIN {X 0,Y 563.634,Z 985.194,A -85,B 0,C 180,E1 24258.975,E2 24258.975} C_VEL
LIN {X 0,Y 559.271,Z 1007.745,A -85,B 0,C 180,E1 24257.344,E2 24257.344} C_VEL
LIN {X 0,Y 554.56,Z 1030.741,A -85,B 0,C 180,E1 24255.412,E2 24255.412} C_VEL
LIN {X 0,Y 549.958,Z 1052.826,A -85,B 0,C 180,E1 24253.268,E2 24253.268} C_VEL
LIN {X 0,Y 545.996,Z 1071.632,A -85,B 0,C 180,E1 24251.177,E2 24251.177} C_VEL
LIN {X 0,Y 541.949,Z 1091.275,A -85,B 0,C 180,E1 24248.7,E2 24248.7} C_VEL
LIN {X 0,Y 538.837,Z 1107.051,A -85,B 0,C 180,E1 24246.426,E2 24246.426} C_VEL
LIN {X 0,Y 536.2,Z 1121.194,A -85,B 0,C 180,E1 24244.144,E2 24244.144} C_VEL
LIN {X 0,Y 533.546,Z 1136.762,A -85,B 0,C 180,E1 24241.271,E2 24241.271} C_VEL
LIN {X 0,Y 531.761,Z 1148.487,A -85,B 0,C 180,E1 24238.774,E2 24238.774} C_VEL
LIN {X 0,Y 530.299,Z 1159.64,A -85,B 0,C 180,E1 24236.06,E2 24236.06} C_VEL
LIN {X 0,Y 529.201,Z 1169.701,A -85,B 0,C 180,E1 24233.141,E2 24233.141} C_VEL
LIN {X 0,Y 528.62,Z 1176.736,A -85,B 0,C 180,E1 24230.714,E2 24230.714} C_VEL
LIN {X 0,Y 528.227,Z 1182.928,A -85,B 0,C 180,E1 24228.149,E2 24228.149} C_VEL
LIN {X 0,Y 528.015,Z 1188.388,A -85,B 0,C 180,E1 24225.261,E2 24225.261} C_VEL
LIN {X 0,Y 527.936,Z 1192.016,A -85,B 0,C 180,E1 24222.469,E2 24222.469} C_VEL
LIN {X 0,Y 527.916,Z 1194.014,A -85,B 0,C 180,E1 24220.035,E2 24220.035} C_VEL
LIN {X 0,Y 527.895,Z 1194.871,A -85,B 0,C 180,E1 24217.619,E2 24217.619} C_VEL
LIN {X 0,Y 527.911,Z 1194.544,A -85,B 0,C 180,E1 24214.78,E2 24214.78} C_VEL
LIN {X 0,Y 527.926,Z 1192.536,A -85,B 0,C 180,E1 24211.954,E2 24211.954} C_VEL
LIN {X 0,Y 527.977,Z 1189.696,A -85,B 0,C 180,E1 24209.566,E2 24209.566} C_VEL
LIN {X 0,Y 528.112,Z 1185.574,A -85,B 0,C 180,E1 24207.07,E2 24207.07} C_VEL
LIN {X 0,Y 528.451,Z 1179.229,A -85,B 0,C 180,E1 24204.136,E2 24204.136} C_VEL
LIN {X 0,Y 529.02,Z 1171.68,A -85,B 0,C 180,E1 24201.413,E2 24201.413} C_VEL
LIN {X 0,Y 529.851,Z 1163.434,A -85,B 0,C 180,E1 24198.903,E2 24198.903} C_VEL
LIN {X 0,Y 531.142,Z 1152.977,A -85,B 0,C 180,E1 24196.168,E2 24196.168} C_VEL
LIN {X 0,Y 532.913,Z 1140.633,A -85,B 0,C 180,E1 24193.43,E2 24193.43} C_VEL
LIN {X 0,Y 534.964,Z 1128.255,A -85,B 0,C 180,E1 24191.022,E2 24191.022} C_VEL
LIN {X 0,Y 537.716,Z 1113.014,A -85,B 0,C 180,E1 24188.397,E2 24188.397} C_VEL
LIN {X 0,Y 540.865,Z 1096.647,A -85,B 0,C 180,E1 24185.959,E2 24185.959} C_VEL
LIN {X 0,Y 543.92,Z 1081.483,A -85,B 0,C 180,E1 24183.938,E2 24183.938} C_VEL
LIN {X 0,Y 547.921,Z 1062.49,A -85,B 0,C 180,E1 24181.676,E2 24181.676} C_VEL
LIN {X 0,Y 552.259,Z 1041.818,A -85,B 0,C 180,E1 24179.54,E2 24179.54} C_VEL
LIN {X 0,Y 556.614,Z 1020.855,A -85,B 0,C 180,E1 24177.636,E2 24177.636} C_VEL
LIN {X 0,Y 561.112,Z 998.272,A -85,B 0,C 180,E1 24175.854,E2 24175.854} C_VEL
LIN {X 0,Y 565.726,Z 974.014,A -85,B 0,C 180,E1 24174.197,E2 24174.197} C_VEL
LIN {X 0,Y 569.709,Z 951.065,A -85,B 0,C 180,E1 24172.863,E2 24172.863} C_VEL
LIN {X 0,Y 573.124,Z 929.905,A -85,B 0,C 180,E1 24171.797,E2 24171.797} C_VEL
LIN {X 0,Y 576.31,Z 908.154,A -85,B 0,C 180,E1 24170.854,E2 24170.854} C_VEL
LIN {X 0,Y 579.85,Z 879.986,A -85,B 0,C 180,E1 24169.85,E2 24169.85} C_VEL
LIN {X 0,Y 582.215,Z 857.101,A -85,B 0,C 180,E1 24169.202,E2 24169.202} C_VEL
LIN {X 0,Y 584.018,Z 835.677,A -85,B 0,C 180,E1 24168.716,E2 24168.716} C_VEL
LIN {X 0,Y 585.422,Z 813.474,A -85,B 0,C 180,E1 24168.328,E2 24168.328} C_VEL
LIN {X 0,Y 592.715,Z 603.849,A -85,B 0,C 180,E1 24165.296,E2 24165.296} C_VEL
LIN {X 0,Y 598.634,Z 437.867,A -85,B 0,C 180,E1 24162.865,E2 24162.865} C_VEL
LIN {X 0,Y 584.049,Z 417.109,A -85,B 0,C 180,E1 24160.552,E2 24160.552} C_VEL
LIN {X 0,Y 572.304,Z 400.806,A -85,B 0,C 180,E1 24158.525,E2 24158.525} C_VEL
LIN {X 0,Y 562.556,Z 388.68,A -85,B 0,C 180,E1 24156.734,E2 24156.734} C_VEL
LIN {X 0,Y 558.089,Z 383.139,A -85,B 0,C 180,E1 24155.864,E2 24155.864} C_VEL
LIN {X 0,Y 553.954,Z 378.055,A -85,B 0,C 180,E1 24155.029,E2 24155.029} C_VEL
LIN {X 0,Y 549.596,Z 372.711,A -85,B 0,C 180,E1 24154.115,E2 24154.115} C_VEL
LIN {X 0,Y 546.068,Z 368.637,A -85,B 0,C 180,E1 24153.352,E2 24153.352} C_VEL
LIN {X 0,Y 544.907,Z 366.971,A -85,B 0,C 180,E1 24153.087,E2 24153.087} C_VEL
LIN {X 0,Y 541.564,Z 363.588,A -85,B 0,C 180,E1 24152.342,E2 24152.342} C_VEL
LIN {X 0,Y 539.847,Z 360.962,A -85,B 0,C 180,E1 24151.924,E2 24151.924} C_VEL
LIN {X 0,Y 536.697,Z 358.123,A -85,B 0,C 180,E1 24151.193,E2 24151.193} C_VEL
LIN {X 0,Y 534.798,Z 354.79,A -85,B 0,C 180,E1 24150.692,E2 24150.692} C_VEL
LIN {X 0,Y 531.708,Z 352.716,A -85,B 0,C 180,E1 24149.953,E2 24149.953} C_VEL
LIN {X 0,Y 530.063,Z 349.929,A -85,B 0,C 180,E1 24149.495,E2 24149.495} C_VEL
LIN {X 0,Y 529.662,Z 348.206,A -85,B 0,C 180,E1 24149.327,E2 24149.327} C_VEL
LIN {X 0,Y 529.599,Z 348.223,A -85,B 0,C 180,E1 24146.017,E2 24146.017} C_VEL
LIN {X 0,Y 529.603,Z 348.194,A -85,B 0,C 180,E1 24142.602,E2 24142.602} C_VEL
LIN {X 0,Y 529.623,Z 348.228,A -85,B 0,C 180,E1 24139.522,E2 24139.522} C_VEL
LIN {X 0,Y 529.6,Z 348.246,A -85,B 0,C 180,E1 24136.226,E2 24136.226} C_VEL
LIN {X 0,Y 529.658,Z 348.237,A -85,B 0,C 180,E1 24133.076,E2 24133.076} C_VEL
LIN {X 0,Y 529.599,Z 348.242,A -85,B 0,C 180,E1 24129.767,E2 24129.767} C_VEL
LIN {X 0,Y 529.645,Z 348.238,A -85,B 0,C 180,E1 24126.504,E2 24126.504} C_VEL
LIN {X 0,Y 529.615,Z 348.246,A -85,B 0,C 180,E1 24123.247,E2 24123.247} C_VEL
LIN {X 0,Y 529.607,Z 348.25,A -85,B 0,C 180,E1 24119.892,E2 24119.892} C_VEL
LIN {X 0,Y 529.659,Z 348.247,A -85,B 0,C 180,E1 24116.645,E2 24116.645} C_VEL
LIN {X 0,Y 529.605,Z 348.261,A -85,B 0,C 180,E1 24113.387,E2 24113.387} C_VEL
LIN {X 0,Y 529.655,Z 348.254,A -85,B 0,C 180,E1 24110.108,E2 24110.108} C_VEL
LIN {X 0,Y 529.614,Z 348.185,A -85,B 0,C 180,E1 24106.795,E2 24106.795} C_VEL
LIN {X 0,Y 529.614,Z 348.254,A -85,B 0,C 180,E1 24103.436,E2 24103.436} C_VEL
LIN {X 0,Y 529.665,Z 348.187,A -85,B 0,C 180,E1 24100.135,E2 24100.135} C_VEL
LIN {X 0,Y 529.686,Z 348.468,A -85,B 0,C 180,E1 24097.741,E2 24097.741} C_VEL
LIN {X 0,Y 530.681,Z 351.335,A -85,B 0,C 180,E1 24097.425,E2 24097.425} C_VEL
LIN {X 0,Y 533.113,Z 353.893,A -85,B 0,C 180,E1 24096.804,E2 24096.804} C_VEL
LIN {X 0,Y 535.081,Z 355.14,A -85,B 0,C 180,E1 24096.341,E2 24096.341} C_VEL
LIN {X 0,Y 537.163,Z 358.688,A -85,B 0,C 180,E1 24095.796,E2 24095.796} C_VEL
LIN {X 0,Y 540.506,Z 361.778,A -85,B 0,C 180,E1 24095.024,E2 24095.024} C_VEL
LIN {X 0,Y 543.594,Z 365.845,A -85,B 0,C 180,E1 24094.301,E2 24094.301} C_VEL
LIN {X 0,Y 549.819,Z 373.479,A -85,B 0,C 180,E1 24092.929,E2 24092.929} C_VEL
LIN {X 0,Y 554.012,Z 378.911,A -85,B 0,C 180,E1 24092.043,E2 24092.043} C_VEL
LIN {X 0,Y 558.883,Z 385.231,A -85,B 0,C 180,E1 24091.056,E2 24091.056} C_VEL
LIN {X 0,Y 568.395,Z 397.837,A -85,B 0,C 180,E1 24089.238,E2 24089.238} C_VEL
LIN {X 0,Y 582.313,Z 417.364,A -85,B 0,C 180,E1 24086.787,E2 24086.787} C_VEL
LIN {X 0,Y 598.495,Z 440.825,A -85,B 0,C 180,E1 24084.201,E2 24084.201} C_VEL
LIN {X 0,Y 598.669,Z 442.169,A -85,B 0,C 180,E1 24084.153,E2 24084.153} C_VEL
LIN {X 0,Y 591.114,Z 654.991,A -85,B 0,C 180,E1 24081.049,E2 24081.049} C_VEL
LIN {X 0,Y 585.144,Z 825.929,A -85,B 0,C 180,E1 24078.574,E2 24078.574} C_VEL
LIN {X 0,Y 583.502,Z 850.065,A -85,B 0,C 180,E1 24078.133,E2 24078.133} C_VEL
LIN {X 0,Y 580.796,Z 878.906,A -85,B 0,C 180,E1 24077.411,E2 24077.411} C_VEL
LIN {X 0,Y 578.249,Z 900.828,A -85,B 0,C 180,E1 24076.715,E2 24076.715} C_VEL
LIN {X 0,Y 575.679,Z 920.394,A -85,B 0,C 180,E1 24075.976,E2 24075.976} C_VEL
LIN {X 0,Y 572.832,Z 939.802,A -85,B 0,C 180,E1 24075.126,E2 24075.126} C_VEL
LIN {X 0,Y 569.572,Z 960.004,A -85,B 0,C 180,E1 24074.11,E2 24074.11} C_VEL
LIN {X 0,Y 565.544,Z 983.351,A -85,B 0,C 180,E1 24072.757,E2 24072.757} C_VEL
LIN {X 0,Y 561.001,Z 1007.39,A -85,B 0,C 180,E1 24071.121,E2 24071.121} C_VEL
LIN {X 0,Y 557.312,Z 1026.055,A -85,B 0,C 180,E1 24069.674,E2 24069.674} C_VEL
LIN {X 0,Y 553.719,Z 1043.77,A -85,B 0,C 180,E1 24068.138,E2 24068.138} C_VEL
LIN {X 0,Y 549.957,Z 1062.203,A -85,B 0,C 180,E1 24066.348,E2 24066.348} C_VEL
LIN {X 0,Y 545.56,Z 1083.532,A -85,B 0,C 180,E1 24063.985,E2 24063.985} C_VEL
LIN {X 0,Y 542.424,Z 1098.822,A -85,B 0,C 180,E1 24062.064,E2 24062.064} C_VEL
LIN {X 0,Y 539.572,Z 1113.062,A -85,B 0,C 180,E1 24060.07,E2 24060.07} C_VEL
LIN {X 0,Y 537.05,Z 1126.47,A -85,B 0,C 180,E1 24057.98,E2 24057.98} C_VEL
LIN {X 0,Y 534.336,Z 1141.972,A -85,B 0,C 180,E1 24055.254,E2 24055.254} C_VEL
LIN {X 0,Y 532.295,Z 1154.742,A -85,B 0,C 180,E1 24052.648,E2 24052.648} C_VEL
LIN {X 0,Y 530.87,Z 1164.978,A -85,B 0,C 180,E1 24050.276,E2 24050.276} C_VEL
LIN {X 0,Y 529.754,Z 1174.321,A -85,B 0,C 180,E1 24047.804,E2 24047.804} C_VEL
LIN {X 0,Y 528.818,Z 1184.246,A -85,B 0,C 180,E1 24044.676,E2 24044.676} C_VEL
LIN {X 0,Y 528.341,Z 1190.819,A -85,B 0,C 180,E1 24042.126,E2 24042.126} C_VEL
LIN {X 0,Y 528.098,Z 1195.905,A -85,B 0,C 180,E1 24039.701,E2 24039.701} C_VEL
LIN {X 0,Y 527.973,Z 1200.003,A -85,B 0,C 180,E1 24037.18,E2 24037.18} C_VEL
LIN {X 0,Y 527.919,Z 1203.273,A -85,B 0,C 180,E1 24034.236,E2 24034.236} C_VEL
LIN {X 0,Y 527.909,Z 1204.69,A -85,B 0,C 180,E1 24031.519,E2 24031.519} C_VEL
LIN {X 0,Y 527.899,Z 1204.849,A -85,B 0,C 180,E1 24029.24,E2 24029.24} C_VEL
LIN {X 0,Y 527.916,Z 1203.969,A -85,B 0,C 180,E1 24026.851,E2 24026.851} C_VEL
LIN {X 0,Y 527.934,Z 1201.977,A -85,B 0,C 180,E1 24024.457,E2 24024.457} C_VEL
LIN {X 0,Y 528.006,Z 1198.724,A -85,B 0,C 180,E1 24021.945,E2 24021.945} C_VEL
LIN {X 0,Y 528.204,Z 1193.351,A -85,B 0,C 180,E1 24018.978,E2 24018.978} C_VEL
LIN {X 0,Y 528.632,Z 1186.669,A -85,B 0,C 180,E1 24016.213,E2 24016.213} C_VEL
LIN {X 0,Y 529.178,Z 1179.857,A -85,B 0,C 180,E1 24013.874,E2 24013.874} C_VEL
LIN {X 0,Y 530.029,Z 1171.89,A -85,B 0,C 180,E1 24011.523,E2 24011.523} C_VEL
LIN {X 0,Y 531.296,Z 1161.771,A -85,B 0,C 180,E1 24008.934,E2 24008.934} C_VEL
LIN {X 0,Y 533.288,Z 1148.285,A -85,B 0,C 180,E1 24005.993,E2 24005.993} C_VEL
LIN {X 0,Y 535.282,Z 1136.327,A -85,B 0,C 180,E1 24003.719,E2 24003.719} C_VEL
LIN {X 0,Y 537.55,Z 1123.669,A -85,B 0,C 180,E1 24001.565,E2 24001.565} C_VEL
LIN {X 0,Y 540.474,Z 1108.747,A -85,B 0,C 180,E1 23999.297,E2 23999.297} C_VEL
LIN {X 0,Y 544.206,Z 1090.047,A -85,B 0,C 180,E1 23996.804,E2 23996.804} C_VEL
LIN {X 0,Y 547.545,Z 1073.682,A -85,B 0,C 180,E1 23994.886,E2 23994.886} C_VEL
LIN {X 0,Y 550.889,Z 1057.429,A -85,B 0,C 180,E1 23993.172,E2 23993.172} C_VEL
LIN {X 0,Y 554.535,Z 1039.706,A -85,B 0,C 180,E1 23991.495,E2 23991.495} C_VEL
LIN {X 0,Y 559.3,Z 1016.182,A -85,B 0,C 180,E1 23989.539,E2 23989.539} C_VEL
LIN {X 0,Y 563.221,Z 995.687,A -85,B 0,C 180,E1 23988.061,E2 23988.061} C_VEL
LIN {X 0,Y 566.639,Z 976.943,A -85,B 0,C 180,E1 23986.862,E2 23986.862} C_VEL
LIN {X 0,Y 570.07,Z 956.897,A -85,B 0,C 180,E1 23985.729,E2 23985.729} C_VEL
LIN {X 0,Y 573.791,Z 933.675,A -85,B 0,C 180,E1 23984.589,E2 23984.589} C_VEL
LIN {X 0,Y 577.548,Z 907.042,A -85,B 0,C 180,E1 23983.5,E2 23983.5} C_VEL
LIN {X 0,Y 580.278,Z 884.677,A -85,B 0,C 180,E1 23982.747,E2 23982.747} C_VEL
LIN {X 0,Y 582.503,Z 863.494,A -85,B 0,C 180,E1 23982.159,E2 23982.159} C_VEL
LIN {X 0,Y 584.39,Z 841.795,A -85,B 0,C 180,E1 23981.679,E2 23981.679} C_VEL
LIN {X 0,Y 586.057,Z 814.587,A -85,B 0,C 180,E1 23981.217,E2 23981.217} C_VEL
LIN {X 0,Y 594.465,Z 591.699,A -85,B 0,C 180,E1 23977.946,E2 23977.946} C_VEL
LIN {X 0,Y 600.614,Z 441.402,A -85,B 0,C 180,E1 23975.698,E2 23975.698} C_VEL
LIN {X 0,Y 591.276,Z 426.526,A -85,B 0,C 180,E1 23973.98,E2 23973.98} C_VEL
LIN {X 0,Y 583.108,Z 414.667,A -85,B 0,C 180,E1 23972.374,E2 23972.374} C_VEL
LIN {X 0,Y 575.124,Z 403.666,A -85,B 0,C 180,E1 23970.682,E2 23970.682} C_VEL
LIN {X 0,Y 568.463,Z 394.833,A -85,B 0,C 180,E1 23969.159,E2 23969.159} C_VEL
LIN {X 0,Y 564.309,Z 389.527,A -85,B 0,C 180,E1 23968.149,E2 23968.149} C_VEL
LIN {X 0,Y 559.573,Z 383.512,A -85,B 0,C 180,E1 23966.929,E2 23966.929} C_VEL
LIN {X 0,Y 554.837,Z 377.65,A -85,B 0,C 180,E1 23965.627,E2 23965.627} C_VEL
LIN {X 0,Y 551.14,Z 373.318,A -85,B 0,C 180,E1 23964.548,E2 23964.548} C_VEL
LIN {X 0,Y 547.8,Z 369.219,A -85,B 0,C 180,E1 23963.505,E2 23963.505} C_VEL
LIN {X 0,Y 546.403,Z 367.655,A -85,B 0,C 180,E1 23963.055,E2 23963.055} C_VEL
LIN {X 0,Y 543.355,Z 364.785,A -85,B 0,C 180,E1 23962.049,E2 23962.049} C_VEL
LIN {X 0,Y 541.465,Z 361.603,A -85,B 0,C 180,E1 23961.333,E2 23961.333} C_VEL
LIN {X 0,Y 538.192,Z 359.432,A -85,B 0,C 180,E1 23960.16,E2 23960.16} C_VEL
LIN {X 0,Y 536.188,Z 356.15,A -85,B 0,C 180,E1 23959.302,E2 23959.302} C_VEL
LIN {X 0,Y 535.693,Z 355.019,A -85,B 0,C 180,E1 23959.065,E2 23959.065} C_VEL
LIN {X 0,Y 532.213,Z 353.119,A -85,B 0,C 180,E1 23957.607,E2 23957.607} C_VEL
LIN {X 0,Y 530.266,Z 350.508,A -85,B 0,C 180,E1 23956.627,E2 23956.627} C_VEL
LIN {X 0,Y 529.648,Z 348.213,A -85,B 0,C 180,E1 23956.168,E2 23956.168} C_VEL
LIN {X 0,Y 529.62,Z 348.204,A -85,B 0,C 180,E1 23952.872,E2 23952.872} C_VEL
LIN {X 0,Y 529.686,Z 348.252,A -85,B 0,C 180,E1 23949.562,E2 23949.562} C_VEL
LIN {X 0,Y 529.621,Z 348.2,A -85,B 0,C 180,E1 23946.287,E2 23946.287} C_VEL
LIN {X 0,Y 529.638,Z 348.222,A -85,B 0,C 180,E1 23942.813,E2 23942.813} C_VEL
LIN {X 0,Y 529.667,Z 348.22,A -85,B 0,C 180,E1 23939.567,E2 23939.567} C_VEL
LIN {X 0,Y 529.621,Z 348.2,A -85,B 0,C 180,E1 23936.211,E2 23936.211} C_VEL
LIN {X 0,Y 529.676,Z 348.251,A -85,B 0,C 180,E1 23932.843,E2 23932.843} C_VEL
LIN {X 0,Y 529.67,Z 348.365,A -85,B 0,C 180,E1 23930.561,E2 23930.561} C_VEL
LIN {X 0,Y 530.443,Z 350.863,A -85,B 0,C 180,E1 23930.068,E2 23930.068} C_VEL
LIN {X 0,Y 532.708,Z 353.541,A -85,B 0,C 180,E1 23928.962,E2 23928.962} C_VEL
LIN {X 0,Y 535.9,Z 355.322,A -85,B 0,C 180,E1 23927.637,E2 23927.637} C_VEL
LIN {X 0,Y 537.574,Z 358.643,A -85,B 0,C 180,E1 23926.884,E2 23926.884} C_VEL
LIN {X 0,Y 540.296,Z 361.053,A -85,B 0,C 180,E1 23925.86,E2 23925.86} C_VEL
LIN {X 0,Y 541.84,Z 361.932,A -85,B 0,C 180,E1 23925.328,E2 23925.328} C_VEL
LIN {X 0,Y 543.932,Z 365.533,A -85,B 0,C 180,E1 23924.541,E2 23924.541} C_VEL
LIN {X 0,Y 547.05,Z 368.039,A -85,B 0,C 180,E1 23923.542,E2 23923.542} C_VEL
LIN {X 0,Y 547.888,Z 369.137,A -85,B 0,C 180,E1 23923.268,E2 23923.268} C_VEL
LIN {X 0,Y 550.616,Z 372.812,A -85,B 0,C 180,E1 23922.401,E2 23922.401} C_VEL
LIN {X 0,Y 553.171,Z 375.002,A -85,B 0,C 180,E1 23921.668,E2 23921.668} C_VEL
LIN {X 0,Y 556.373,Z 379.232,A -85,B 0,C 180,E1 23920.745,E2 23920.745} C_VEL
LIN {X 0,Y 558.545,Z 381.302,A -85,B 0,C 180,E1 23920.169,E2 23920.169} C_VEL
LIN {X 0,Y 562.17,Z 385.805,A -85,B 0,C 180,E1 23919.216,E2 23919.216} C_VEL
LIN {X 0,Y 563.961,Z 387.847,A -85,B 0,C 180,E1 23918.769,E2 23918.769} C_VEL
LIN {X 0,Y 568.787,Z 393.721,A -85,B 0,C 180,E1 23917.602,E2 23917.602} C_VEL
LIN {X 0,Y 573.819,Z 399.954,A -85,B 0,C 180,E1 23916.455,E2 23916.455} C_VEL
LIN {X 0,Y 580.124,Z 407.898,A -85,B 0,C 180,E1 23915.103,E2 23915.103} C_VEL
LIN {X 0,Y 589.89,Z 421.651,A -85,B 0,C 180,E1 23913.145,E2 23913.145} C_VEL
LIN {X 0,Y 598.286,Z 434.488,A -85,B 0,C 180,E1 23911.582,E2 23911.582} C_VEL
LIN {X 0,Y 600.564,Z 438.474,A -85,B 0,C 180,E1 23911.168,E2 23911.168} C_VEL
LIN {X 0,Y 591.91,Z 652.057,A -85,B 0,C 180,E1 23907.984,E2 23907.984} C_VEL
LIN {X 0,Y 585.52,Z 818.11,A -85,B 0,C 180,E1 23905.537,E2 23905.537} C_VEL
LIN {X 0,Y 583.736,Z 843.372,A -85,B 0,C 180,E1 23905.061,E2 23905.061} C_VEL
LIN {X 0,Y 581.034,Z 870.748,A -85,B 0,C 180,E1 23904.356,E2 23904.356} C_VEL
LIN {X 0,Y 578.455,Z 892.411,A -85,B 0,C 180,E1 23903.656,E2 23903.656} C_VEL
LIN {X 0,Y 575.679,Z 913.002,A -85,B 0,C 180,E1 23902.864,E2 23902.864} C_VEL
LIN {X 0,Y 574.961,Z 918.119,A -85,B 0,C 180,E1 23902.651,E2 23902.651} C_VEL
LIN {X 0,Y 573.222,Z 925.314,A -85,B 0,C 180,E1 23902.409,E2 23902.409} C_VEL
LIN {X 0,Y 565.955,Z 943.633,A -85,B 0,C 180,E1 23901.962,E2 23901.962} C_VEL
LIN {X 0,Y 564.019,Z 950.451,A -85,B 0,C 180,E1 23901.669,E2 23901.669} C_VEL
LIN {X 0,Y 559.958,Z 972.725,A -85,B 0,C 180,E1 23900.368,E2 23900.368} C_VEL
LIN {X 0,Y 555.084,Z 997.389,A -85,B 0,C 180,E1 23898.688,E2 23898.688} C_VEL
LIN {X 0,Y 550.886,Z 1017.548,A -85,B 0,C 180,E1 23897.105,E2 23897.105} C_VEL
LIN {X 0,Y 546.352,Z 1038.849,A -85,B 0,C 180,E1 23895.203,E2 23895.203} C_VEL
LIN {X 0,Y 541.701,Z 1059.967,A -85,B 0,C 180,E1 23893.033,E2 23893.033} C_VEL
LIN {X 0,Y 537.111,Z 1080.684,A -85,B 0,C 180,E1 23890.576,E2 23890.576} C_VEL
LIN {X 0,Y 533.662,Z 1096.798,A -85,B 0,C 180,E1 23888.396,E2 23888.396} C_VEL
LIN {X 0,Y 530.162,Z 1114.033,A -85,B 0,C 180,E1 23885.778,E2 23885.778} C_VEL
LIN {X 0,Y 527.373,Z 1128.587,A -85,B 0,C 180,E1 23883.224,E2 23883.224} C_VEL
LIN {X 0,Y 525.248,Z 1140.835,A -85,B 0,C 180,E1 23880.801,E2 23880.801} C_VEL
LIN {X 0,Y 523.301,Z 1153.592,A -85,B 0,C 180,E1 23877.912,E2 23877.912} C_VEL
LIN {X 0,Y 521.949,Z 1163.848,A -85,B 0,C 180,E1 23875.168,E2 23875.168} C_VEL
LIN {X 0,Y 521.071,Z 1172.194,A -85,B 0,C 180,E1 23872.567,E2 23872.567} C_VEL
LIN {X 0,Y 520.413,Z 1180.267,A -85,B 0,C 180,E1 23869.53,E2 23869.53} C_VEL
LIN {X 0,Y 520.119,Z 1185.938,A -85,B 0,C 180,E1 23866.789,E2 23866.789} C_VEL
LIN {X 0,Y 519.984,Z 1189.826,A -85,B 0,C 180,E1 23864.362,E2 23864.362} C_VEL
LIN {X 0,Y 519.921,Z 1192.804,A -85,B 0,C 180,E1 23861.762,E2 23861.762} C_VEL
LIN {X 0,Y 519.91,Z 1194.626,A -85,B 0,C 180,E1 23858.85,E2 23858.85} C_VEL
LIN {X 0,Y 519.913,Z 1194.852,A -85,B 0,C 180,E1 23856.182,E2 23856.182} C_VEL
LIN {X 0,Y 519.908,Z 1193.965,A -85,B 0,C 180,E1 23853.749,E2 23853.749} C_VEL
LIN {X 0,Y 519.933,Z 1191.98,A -85,B 0,C 180,E1 23851.322,E2 23851.322} C_VEL
LIN {X 0,Y 520.02,Z 1188.458,A -85,B 0,C 180,E1 23848.568,E2 23848.568} C_VEL
LIN {X 0,Y 520.252,Z 1182.934,A -85,B 0,C 180,E1 23845.591,E2 23845.591} C_VEL
LIN {X 0,Y 520.664,Z 1176.915,A -85,B 0,C 180,E1 23843.051,E2 23843.051} C_VEL
LIN {X 0,Y 521.32,Z 1169.666,A -85,B 0,C 180,E1 23840.506,E2 23840.506} C_VEL
LIN {X 0,Y 522.552,Z 1159.002,A -85,B 0,C 180,E1 23837.39,E2 23837.39} C_VEL
LIN {X 0,Y 524.063,Z 1148.206,A -85,B 0,C 180,E1 23834.735,E2 23834.735} C_VEL
LIN {X 0,Y 525.998,Z 1136.349,A -85,B 0,C 180,E1 23832.179,E2 23832.179} C_VEL
LIN {X 0,Y 528.826,Z 1120.855,A -85,B 0,C 180,E1 23829.295,E2 23829.295} C_VEL
LIN {X 0,Y 531.46,Z 1107.328,A -85,B 0,C 180,E1 23827.081,E2 23827.081} C_VEL
LIN {X 0,Y 534.955,Z 1090.77,A -85,B 0,C 180,E1 23824.659,E2 23824.659} C_VEL
LIN {X 0,Y 539.126,Z 1071.546,A -85,B 0,C 180,E1 23822.211,E2 23822.211} C_VEL
LIN {X 0,Y 543.534,Z 1051.555,A -85,B 0,C 180,E1 23819.976,E2 23819.976} C_VEL
LIN {X 0,Y 548.368,Z 1029.411,A -85,B 0,C 180,E1 23817.831,E2 23817.831} C_VEL
LIN {X 0,Y 553.49,Z 1005.286,A -85,B 0,C 180,E1 23815.819,E2 23815.819} C_VEL
LIN {X 0,Y 557.571,Z 984.995,A -85,B 0,C 180,E1 23814.352,E2 23814.352} C_VEL
LIN {X 0,Y 561.146,Z 966.253,A -85,B 0,C 180,E1 23813.154,E2 23813.154} C_VEL
LIN {X 0,Y 564.701,Z 946.29,A -85,B 0,C 180,E1 23812.028,E2 23812.028} C_VEL
LIN {X 0,Y 568.805,Z 921.125,A -85,B 0,C 180,E1 23810.807,E2 23810.807} C_VEL
LIN {X 0,Y 572.259,Z 896.351,A -85,B 0,C 180,E1 23809.823,E2 23809.823} C_VEL
LIN {X 0,Y 574.861,Z 874.952,A -85,B 0,C 180,E1 23809.113,E2 23809.113} C_VEL
LIN {X 0,Y 577.032,Z 853.948,A -85,B 0,C 180,E1 23808.538,E2 23808.538} C_VEL
LIN {X 0,Y 578.972,Z 831.06,A -85,B 0,C 180,E1 23808.041,E2 23808.041} C_VEL
LIN {X 0,Y 580.794,Z 795.32,A -85,B 0,C 180,E1 23807.47,E2 23807.47} C_VEL
LIN {X 0,Y 588.746,Z 572.737,A -85,B 0,C 180,E1 23804.241,E2 23804.241} C_VEL
LIN {X 0,Y 593.52,Z 441.933,A -85,B 0,C 180,E1 23802.302,E2 23802.302} C_VEL
LIN {X 0,Y 577.369,Z 418.837,A -85,B 0,C 180,E1 23799.656,E2 23799.656} C_VEL
LIN {X 0,Y 568.408,Z 406.589,A -85,B 0,C 180,E1 23798.066,E2 23798.066} C_VEL
LIN {X 0,Y 559.624,Z 395.453,A -85,B 0,C 180,E1 23796.416,E2 23796.416} C_VEL
LIN {X 0,Y 555.083,Z 389.791,A -85,B 0,C 180,E1 23795.516,E2 23795.516} C_VEL
LIN {X 0,Y 551.104,Z 384.874,A -85,B 0,C 180,E1 23794.698,E2 23794.698} C_VEL
LIN {X 0,Y 546.778,Z 379.588,A -85,B 0,C 180,E1 23793.775,E2 23793.775} C_VEL
LIN {X 0,Y 543.107,Z 375.071,A -85,B 0,C 180,E1 23792.959,E2 23792.959} C_VEL
LIN {X 0,Y 538.563,Z 369.891,A -85,B 0,C 180,E1 23791.915,E2 23791.915} C_VEL
LIN {X 0,Y 537.245,Z 368.117,A -85,B 0,C 180,E1 23791.595,E2 23791.595} C_VEL
LIN {X 0,Y 533.965,Z 364.754,A -85,B 0,C 180,E1 23790.807,E2 23790.807} C_VEL
LIN {X 0,Y 532.239,Z 362.131,A -85,B 0,C 180,E1 23790.355,E2 23790.355} C_VEL
LIN {X 0,Y 529.043,Z 359.423,A -85,B 0,C 180,E1 23789.557,E2 23789.557} C_VEL
LIN {X 0,Y 526.891,Z 355.721,A -85,B 0,C 180,E1 23788.942,E2 23788.942} C_VEL
LIN {X 0,Y 523.752,Z 353.656,A -85,B 0,C 180,E1 23788.119,E2 23788.119} C_VEL
LIN {X 0,Y 522.089,Z 350.856,A -85,B 0,C 180,E1 23787.612,E2 23787.612} C_VEL
LIN {X 0,Y 521.714,Z 349.172,A -85,B 0,C 180,E1 23787.423,E2 23787.423} C_VEL
LIN {X 0,Y 521.657,Z 349.232,A -85,B 0,C 180,E1 23784.096,E2 23784.096} C_VEL
LIN {X 0,Y 521.679,Z 349.178,A -85,B 0,C 180,E1 23780.723,E2 23780.723} C_VEL
LIN {X 0,Y 521.684,Z 349.236,A -85,B 0,C 180,E1 23777.513,E2 23777.513} C_VEL
LIN {X 0,Y 521.662,Z 349.241,A -85,B 0,C 180,E1 23774.202,E2 23774.202} C_VEL
LIN {X 0,Y 521.722,Z 349.236,A -85,B 0,C 180,E1 23770.937,E2 23770.937} C_VEL
LIN {X 0,Y 521.667,Z 349.25,A -85,B 0,C 180,E1 23767.6,E2 23767.6} C_VEL
LIN {X 0,Y 521.682,Z 349.247,A -85,B 0,C 180,E1 23764.177,E2 23764.177} C_VEL
LIN {X 0,Y 521.708,Z 349.246,A -85,B 0,C 180,E1 23760.879,E2 23760.879} C_VEL
LIN {X 0,Y 521.666,Z 349.25,A -85,B 0,C 180,E1 23757.583,E2 23757.583} C_VEL
LIN {X 0,Y 521.722,Z 349.237,A -85,B 0,C 180,E1 23754.28,E2 23754.28} C_VEL
LIN {X 0,Y 521.672,Z 349.241,A -85,B 0,C 180,E1 23751.068,E2 23751.068} C_VEL
LIN {X 0,Y 521.669,Z 349.174,A -85,B 0,C 180,E1 23747.604,E2 23747.604} C_VEL
LIN {X 0,Y 521.726,Z 349.238,A -85,B 0,C 180,E1 23744.322,E2 23744.322} C_VEL
LIN {X 0,Y 521.663,Z 349.177,A -85,B 0,C 180,E1 23740.983,E2 23740.983} C_VEL
LIN {X 0,Y 521.703,Z 349.275,A -85,B 0,C 180,E1 23739.643,E2 23739.643} C_VEL
LIN {X 0,Y 522.583,Z 352.038,A -85,B 0,C 180,E1 23739.328,E2 23739.328} C_VEL
LIN {X 0,Y 524.92,Z 354.712,A -85,B 0,C 180,E1 23738.665,E2 23738.665} C_VEL
LIN {X 0,Y 527.208,Z 356.101,A -85,B 0,C 180,E1 23738.075,E2 23738.075} C_VEL
LIN {X 0,Y 529.2,Z 359.628,A -85,B 0,C 180,E1 23737.504,E2 23737.504} C_VEL
LIN {X 0,Y 532.503,Z 362.203,A -85,B 0,C 180,E1 23736.688,E2 23736.688} C_VEL
LIN {X 0,Y 535.278,Z 366.372,A -85,B 0,C 180,E1 23735.97,E2 23735.97} C_VEL
LIN {X 0,Y 538.074,Z 368.976,A -85,B 0,C 180,E1 23735.314,E2 23735.314} C_VEL
LIN {X 0,Y 541.459,Z 373.287,A -85,B 0,C 180,E1 23734.515,E2 23734.515} C_VEL
LIN {X 0,Y 550.365,Z 384.483,A -85,B 0,C 180,E1 23732.548,E2 23732.548} C_VEL
LIN {X 0,Y 562.183,Z 400.154,A -85,B 0,C 180,E1 23730.161,E2 23730.161} C_VEL
LIN {X 0,Y 574.304,Z 417.197,A -85,B 0,C 180,E1 23727.925,E2 23727.925} C_VEL
LIN {X 0,Y 589,Z 438.364,A -85,B 0,C 180,E1 23725.458,E2 23725.458} C_VEL
LIN {X 0,Y 593.656,Z 445.461,A -85,B 0,C 180,E1 23724.717,E2 23724.717} C_VEL
LIN {X 0,Y 585.74,Z 660.178,A -85,B 0,C 180,E1 23721.571,E2 23721.571} C_VEL
LIN {X 0,Y 579.736,Z 826.004,A -85,B 0,C 180,E1 23719.157,E2 23719.157} C_VEL
LIN {X 0,Y 578,Z 850.694,A -85,B 0,C 180,E1 23718.703,E2 23718.703} C_VEL
LIN {X 0,Y 575.249,Z 878.954,A -85,B 0,C 180,E1 23717.992,E2 23717.992} C_VEL
LIN {X 0,Y 572.586,Z 901.174,A -85,B 0,C 180,E1 23717.283,E2 23717.283} C_VEL
LIN {X 0,Y 569.75,Z 921.97,A -85,B 0,C 180,E1 23716.49,E2 23716.49} C_VEL
LIN {X 0,Y 566.717,Z 941.871,A -85,B 0,C 180,E1 23715.605,E2 23715.605} C_VEL
LIN {X 0,Y 562.694,Z 965.924,A -85,B 0,C 180,E1 23714.364,E2 23714.364} C_VEL
LIN {X 0,Y 558.203,Z 989.933,A -85,B 0,C 180,E1 23712.893,E2 23712.893} C_VEL
LIN {X 0,Y 554.355,Z 1009.283,A -85,B 0,C 180,E1 23711.536,E2 23711.536} C_VEL
LIN {X 0,Y 550.537,Z 1027.762,A -85,B 0,C 180,E1 23710.077,E2 23710.077} C_VEL
LIN {X 0,Y 546.409,Z 1047.331,A -85,B 0,C 180,E1 23708.34,E2 23708.34} C_VEL
LIN {X 0,Y 541.602,Z 1069.514,A -85,B 0,C 180,E1 23706.079,E2 23706.079} C_VEL
LIN {X 0,Y 538.127,Z 1085.577,A -85,B 0,C 180,E1 23704.223,E2 23704.223} C_VEL
LIN {X 0,Y 534.949,Z 1100.454,A -85,B 0,C 180,E1 23702.314,E2 23702.314} C_VEL
LIN {X 0,Y 532.097,Z 1114.139,A -85,B 0,C 180,E1 23700.363,E2 23700.363} C_VEL
LIN {X 0,Y 528.99,Z 1130.164,A -85,B 0,C 180,E1 23697.796,E2 23697.796} C_VEL
LIN {X 0,Y 526.245,Z 1144.838,A -85,B 0,C 180,E1 23695.068,E2 23695.068} C_VEL
LIN {X 0,Y 524.441,Z 1155.769,A -85,B 0,C 180,E1 23692.769,E2 23692.769} C_VEL
LIN {X 0,Y 522.963,Z 1165.895,A -85,B 0,C 180,E1 23690.363,E2 23690.363} C_VEL
LIN {X 0,Y 521.631,Z 1176.674,A -85,B 0,C 180,E1 23687.399,E2 23687.399} C_VEL
LIN {X 0,Y 520.805,Z 1185.152,A -85,B 0,C 180,E1 23684.566,E2 23684.566} C_VEL
LIN {X 0,Y 520.345,Z 1191.325,A -85,B 0,C 180,E1 23682.09,E2 23682.09} C_VEL
LIN {X 0,Y 520.088,Z 1196.542,A -85,B 0,C 180,E1 23679.506,E2 23679.506} C_VEL
LIN {X 0,Y 519.955,Z 1201.053,A -85,B 0,C 180,E1 23676.514,E2 23676.514} C_VEL
LIN {X 0,Y 519.913,Z 1203.627,A -85,B 0,C 180,E1 23673.749,E2 23673.749} C_VEL
LIN {X 0,Y 519.914,Z 1204.735,A -85,B 0,C 180,E1 23671.322,E2 23671.322} C_VEL
LIN {X 0,Y 519.909,Z 1204.803,A -85,B 0,C 180,E1 23669.008,E2 23669.008} C_VEL
LIN {X 0,Y 519.916,Z 1203.898,A -85,B 0,C 180,E1 23666.693,E2 23666.693} C_VEL
LIN {X 0,Y 519.937,Z 1201.861,A -85,B 0,C 180,E1 23664.261,E2 23664.261} C_VEL
LIN {X 0,Y 520.022,Z 1198.401,A -85,B 0,C 180,E1 23661.597,E2 23661.597} C_VEL
LIN {X 0,Y 520.256,Z 1192.832,A -85,B 0,C 180,E1 23658.575,E2 23658.575} C_VEL
LIN {X 0,Y 520.713,Z 1186.309,A -85,B 0,C 180,E1 23655.865,E2 23655.865} C_VEL
LIN {X 0,Y 521.322,Z 1179.503,A -85,B 0,C 180,E1 23653.51,E2 23653.51} C_VEL
LIN {X 0,Y 522.275,Z 1171.205,A -85,B 0,C 180,E1 23651.043,E2 23651.043} C_VEL
LIN {X 0,Y 523.851,Z 1159.893,A -85,B 0,C 180,E1 23648.149,E2 23648.149} C_VEL
LIN {X 0,Y 525.859,Z 1147.136,A -85,B 0,C 180,E1 23645.392,E2 23645.392} C_VEL
LIN {X 0,Y 527.943,Z 1135.319,A -85,B 0,C 180,E1 23643.132,E2 23643.132} C_VEL
LIN {X 0,Y 530.483,Z 1122.266,A -85,B 0,C 180,E1 23640.904,E2 23640.904} C_VEL
LIN {X 0,Y 534.082,Z 1104.701,A -85,B 0,C 180,E1 23638.26,E2 23638.26} C_VEL
LIN {X 0,Y 537.638,Z 1087.753,A -85,B 0,C 180,E1 23636.044,E2 23636.044} C_VEL
LIN {X 0,Y 540.955,Z 1072.347,A -85,B 0,C 180,E1 23634.237,E2 23634.237} C_VEL
LIN {X 0,Y 544.638,Z 1055.368,A -85,B 0,C 180,E1 23632.447,E2 23632.447} C_VEL
LIN {X 0,Y 549.329,Z 1033.739,A -85,B 0,C 180,E1 23630.428,E2 23630.428} C_VEL
LIN {X 0,Y 553.741,Z 1012.246,A -85,B 0,C 180,E1 23628.692,E2 23628.692} C_VEL
LIN {X 0,Y 557.421,Z 993.807,A -85,B 0,C 180,E1 23627.373,E2 23627.373} C_VEL
LIN {X 0,Y 560.976,Z 975.133,A -85,B 0,C 180,E1 23626.183,E2 23626.183} C_VEL
LIN {X 0,Y 564.604,Z 954.89,A -85,B 0,C 180,E1 23625.042,E2 23625.042} C_VEL
LIN {X 0,Y 568.795,Z 929.61,A -85,B 0,C 180,E1 23623.814,E2 23623.814} C_VEL
LIN {X 0,Y 572.307,Z 905.13,A -85,B 0,C 180,E1 23622.834,E2 23622.834} C_VEL
LIN {X 0,Y 575.016,Z 883.844,A -85,B 0,C 180,E1 23622.122,E2 23622.122} C_VEL
LIN {X 0,Y 577.319,Z 862.608,A -85,B 0,C 180,E1 23621.534,E2 23621.534} C_VEL
LIN {X 0,Y 579.316,Z 840.368,A -85,B 0,C 180,E1 23621.047,E2 23621.047} C_VEL
LIN {X 0,Y 581.121,Z 809.646,A -85,B 0,C 180,E1 23620.538,E2 23620.538} C_VEL
LIN {X 0,Y 590.074,Z 584.122,A -85,B 0,C 180,E1 23617.203,E2 23617.203} C_VEL
LIN {X 0,Y 595.943,Z 445.39,A -85,B 0,C 180,E1 23615.105,E2 23615.105} C_VEL
LIN {X 0,Y 585.893,Z 429.465,A -85,B 0,C 180,E1 23613.189,E2 23613.189} C_VEL
LIN {X 0,Y 576.456,Z 415.952,A -85,B 0,C 180,E1 23611.241,E2 23611.241} C_VEL
LIN {X 0,Y 566.825,Z 402.782,A -85,B 0,C 180,E1 23609.048,E2 23609.048} C_VEL
LIN {X 0,Y 561.694,Z 396.319,A -85,B 0,C 180,E1 23607.786,E2 23607.786} C_VEL
LIN {X 0,Y 557.19,Z 390.514,A -85,B 0,C 180,E1 23606.598,E2 23606.598} C_VEL
LIN {X 0,Y 552.683,Z 384.85,A -85,B 0,C 180,E1 23605.332,E2 23605.332} C_VEL
LIN {X 0,Y 549.203,Z 380.73,A -85,B 0,C 180,E1 23604.297,E2 23604.297} C_VEL
LIN {X 0,Y 545.536,Z 376.066,A -85,B 0,C 180,E1 23603.122,E2 23603.122} C_VEL
LIN {X 0,Y 541.534,Z 372.163,A -85,B 0,C 180,E1 23601.785,E2 23601.785} C_VEL
LIN {X 0,Y 539.944,Z 369.371,A -85,B 0,C 180,E1 23601.168,E2 23601.168} C_VEL
LIN {X 0,Y 536.581,Z 366.992,A -85,B 0,C 180,E1 23599.939,E2 23599.939} C_VEL
LIN {X 0,Y 534.434,Z 363.452,A -85,B 0,C 180,E1 23598.999,E2 23598.999} C_VEL
LIN {X 0,Y 533.968,Z 362.755,A -85,B 0,C 180,E1 23598.789,E2 23598.789} C_VEL
LIN {X 0,Y 530.472,Z 360.511,A -85,B 0,C 180,E1 23597.27,E2 23597.27} C_VEL
LIN {X 0,Y 528.563,Z 357.568,A -85,B 0,C 180,E1 23596.259,E2 23596.259} C_VEL
LIN {X 0,Y 528.068,Z 356.053,A -85,B 0,C 180,E1 23595.936,E2 23595.936} C_VEL
LIN {X 0,Y 524.733,Z 354.545,A -85,B 0,C 180,E1 23594.117,E2 23594.117} C_VEL
LIN {X 0,Y 522.363,Z 351.566,A -85,B 0,C 180,E1 23592.436,E2 23592.436} C_VEL
LIN {X 0,Y 521.737,Z 349.181,A -85,B 0,C 180,E1 23591.721,E2 23591.721} C_VEL
LIN {X 0,Y 521.683,Z 349.215,A -85,B 0,C 180,E1 23588.487,E2 23588.487} C_VEL
LIN {X 0,Y 521.723,Z 349.204,A -85,B 0,C 180,E1 23585.168,E2 23585.168} C_VEL
LIN {X 0,Y 521.7,Z 349.187,A -85,B 0,C 180,E1 23581.867,E2 23581.867} C_VEL
LIN {X 0,Y 521.692,Z 349.249,A -85,B 0,C 180,E1 23578.462,E2 23578.462} C_VEL
LIN {X 0,Y 521.738,Z 349.182,A -85,B 0,C 180,E1 23575.163,E2 23575.163} C_VEL
LIN {X 0,Y 521.779,Z 349.523,A -85,B 0,C 180,E1 23574.943,E2 23574.943} C_VEL
LIN {X 0,Y 522.642,Z 352.13,A -85,B 0,C 180,E1 23574.125,E2 23574.125} C_VEL
LIN {X 0,Y 525.47,Z 355.066,A -85,B 0,C 180,E1 23572.235,E2 23572.235} C_VEL
LIN {X 0,Y 528.165,Z 356.331,A -85,B 0,C 180,E1 23570.795,E2 23570.795} C_VEL
LIN {X 0,Y 529.528,Z 359.373,A -85,B 0,C 180,E1 23569.996,E2 23569.996} C_VEL
LIN {X 0,Y 532.697,Z 362.225,A -85,B 0,C 180,E1 23568.523,E2 23568.523} C_VEL
LIN {X 0,Y 534.331,Z 363.177,A -85,B 0,C 180,E1 23567.847,E2 23567.847} C_VEL
LIN {X 0,Y 536.447,Z 366.803,A -85,B 0,C 180,E1 23566.911,E2 23566.911} C_VEL
LIN {X 0,Y 539.631,Z 369.219,A -85,B 0,C 180,E1 23565.733,E2 23565.733} C_VEL
LIN {X 0,Y 540.316,Z 370.05,A -85,B 0,C 180,E1 23565.478,E2 23565.478} C_VEL
